LIN {X 0,Y 539.411,Z 297.162,A -85,B 0,C 180,E1 -4153.42,E2 -4153.42} C_VEL
LIN {X 0,Y 539.753,Z 202.979,A -85,B 0,C 180,E1 -4154.735,E2 -4154.735} C_VEL
LIN {X 0,Y 538.601,Z 196.337,A -85,B 0,C 180,E1 -4154.875,E2 -4154.875} C_VEL
LIN {X 0,Y 538.99,Z 174.234,A -85,B 0,C 180,E1 -4158.237,E2 -4158.237} C_VEL
LIN {X 0,Y 539.44,Z 154.956,A -85,B 0,C 180,E1 -4161.195,E2 -4161.195} C_VEL
LIN {X 0,Y 539.677,Z 143.31,A -85,B 0,C 180,E1 -4162.997,E2 -4162.997} C_VEL
LIN {X 0,Y 539.202,Z 140.592,A -85,B 0,C 180,E1 -4163.445,E2 -4163.445} C_VEL
LIN {X 0,Y 538.106,Z 138.749,A -85,B 0,C 180,E1 -4163.808,E2 -4163.808} C_VEL
LIN {X 0,Y 536.213,Z 137.465,A -85,B 0,C 180,E1 -4164.169,E2 -4164.169} C_VEL
LIN {X 0,Y 532.769,Z 136.298,A -85,B 0,C 180,E1 -4164.789,E2 -4164.789} C_VEL
LIN {X 0,Y 531.182,Z 135.998,A -85,B 0,C 180,E1 -4165.267,E2 -4165.267} C_VEL
LIN {X 0,Y 530.982,Z 135.97,A -85,B 0,C 180,E1 -4165.483,E2 -4165.483} C_VEL
LIN {X 0,Y 530.969,Z 135.967,A -85,B 0,C 180,E1 -4168.457,E2 -4168.457} C_VEL
LIN {X 0,Y 530.958,Z 135.972,A -85,B 0,C 180,E1 -4171.079,E2 -4171.079} C_VEL
LIN {X 0,Y 530.991,Z 135.967,A -85,B 0,C 180,E1 -4173.773,E2 -4173.773} C_VEL
LIN {X 0,Y 530.955,Z 135.968,A -85,B 0,C 180,E1 -4176.559,E2 -4176.559} C_VEL
LIN {X 0,Y 530.989,Z 135.966,A -85,B 0,C 180,E1 -4179.443,E2 -4179.443} C_VEL
LIN {X 0,Y 530.968,Z 135.967,A -85,B 0,C 180,E1 -4182.458,E2 -4182.458} C_VEL
LIN {X 0,Y 530.986,Z 135.965,A -85,B 0,C 180,E1 -4185.621,E2 -4185.621} C_VEL
LIN {X 0,Y 530.998,Z 135.966,A -85,B 0,C 180,E1 -4188.564,E2 -4188.564} C_VEL
LIN {X 0,Y 530.96,Z 135.97,A -85,B 0,C 180,E1 -4191.529,E2 -4191.529} C_VEL
LIN {X 0,Y 530.958,Z 135.972,A -85,B 0,C 180,E1 -4194.379,E2 -4194.379} C_VEL
LIN {X 0,Y 530.971,Z 135.971,A -85,B 0,C 180,E1 -4197.133,E2 -4197.133} C_VEL
LIN {X 0,Y 530.965,Z 135.968,A -85,B 0,C 180,E1 -4199.802,E2 -4199.802} C_VEL
LIN {X 0,Y 531.015,Z 135.969,A -85,B 0,C 180,E1 -4202.467,E2 -4202.467} C_VEL
LIN {X 0,Y 531.02,Z 136.091,A -85,B 0,C 180,E1 -4205.464,E2 -4205.464} C_VEL
LIN {X 0,Y 532.94,Z 145.226,A -85,B 0,C 180,E1 -4206.9,E2 -4206.9} C_VEL
LIN {X 0,Y 532.794,Z 159.001,A -85,B 0,C 180,E1 -4208.844,E2 -4208.844} C_VEL
LIN {X 0,Y 535.286,Z 169.811,A -85,B 0,C 180,E1 -4209.115,E2 -4209.115} C_VEL
LIN {X 0,Y 534.354,Z 324.425,A -85,B 0,C 180,E1 -4211.272,E2 -4211.272} C_VEL
LIN {X 0,Y 534.175,Z 339.836,A -85,B 0,C 180,E1 -4211.642,E2 -4211.642} C_VEL
LIN {X 0,Y 533.837,Z 353.957,A -85,B 0,C 180,E1 -4212.126,E2 -4212.126} C_VEL
LIN {X 0,Y 533.535,Z 367.904,A -85,B 0,C 180,E1 -4212.759,E2 -4212.759} C_VEL
LIN {X 0,Y 533.102,Z 381.485,A -85,B 0,C 180,E1 -4213.534,E2 -4213.534} C_VEL
LIN {X 0,Y 532.63,Z 394.075,A -85,B 0,C 180,E1 -4214.414,E2 -4214.414} C_VEL
LIN {X 0,Y 532.206,Z 406.499,A -85,B 0,C 180,E1 -4215.468,E2 -4215.468} C_VEL
LIN {X 0,Y 531.807,Z 417.877,A -85,B 0,C 180,E1 -4216.627,E2 -4216.627} C_VEL
LIN {X 0,Y 531.428,Z 427.452,A -85,B 0,C 180,E1 -4217.783,E2 -4217.783} C_VEL
LIN {X 0,Y 531.172,Z 436.798,A -85,B 0,C 180,E1 -4219.131,E2 -4219.131} C_VEL
LIN {X 0,Y 530.874,Z 444.587,A -85,B 0,C 180,E1 -4220.474,E2 -4220.474} C_VEL
LIN {X 0,Y 530.694,Z 451.826,A -85,B 0,C 180,E1 -4222.006,E2 -4222.006} C_VEL
LIN {X 0,Y 530.578,Z 457.254,A -85,B 0,C 180,E1 -4223.437,E2 -4223.437} C_VEL
LIN {X 0,Y 530.52,Z 460.953,A -85,B 0,C 180,E1 -4224.678,E2 -4224.678} C_VEL
LIN {X 0,Y 530.513,Z 464.408,A -85,B 0,C 180,E1 -4226.201,E2 -4226.201} C_VEL
LIN {X 0,Y 530.416,Z 466.698,A -85,B 0,C 180,E1 -4227.721,E2 -4227.721} C_VEL
LIN {X 0,Y 530.364,Z 467.866,A -85,B 0,C 180,E1 -4229.24,E2 -4229.24} C_VEL
LIN {X 0,Y 530.364,Z 467.884,A -85,B 0,C 180,E1 -4230.758,E2 -4230.758} C_VEL
LIN {X 0,Y 530.416,Z 466.787,A -85,B 0,C 180,E1 -4232.277,E2 -4232.277} C_VEL
LIN {X 0,Y 530.513,Z 464.572,A -85,B 0,C 180,E1 -4233.797,E2 -4233.797} C_VEL
LIN {X 0,Y 530.519,Z 461.201,A -85,B 0,C 180,E1 -4235.32,E2 -4235.32} C_VEL
LIN {X 0,Y 530.603,Z 456.572,A -85,B 0,C 180,E1 -4236.845,E2 -4236.845} C_VEL
LIN {X 0,Y 530.762,Z 450.558,A -85,B 0,C 180,E1 -4238.374,E2 -4238.374} C_VEL
LIN {X 0,Y 530.907,Z 442.996,A -85,B 0,C 180,E1 -4239.908,E2 -4239.908} C_VEL
LIN {X 0,Y 531.198,Z 434.918,A -85,B 0,C 180,E1 -4241.252,E2 -4241.252} C_VEL
LIN {X 0,Y 531.528,Z 425.173,A -85,B 0,C 180,E1 -4242.6,E2 -4242.6} C_VEL
LIN {X 0,Y 531.895,Z 415.216,A -85,B 0,C 180,E1 -4243.758,E2 -4243.758} C_VEL
LIN {X 0,Y 532.319,Z 403.281,A -85,B 0,C 180,E1 -4244.918,E2 -4244.918} C_VEL
LIN {X 0,Y 532.784,Z 391.316,A -85,B 0,C 180,E1 -4245.886,E2 -4245.886} C_VEL
LIN {X 0,Y 533.207,Z 378.321,A -85,B 0,C 180,E1 -4246.757,E2 -4246.757} C_VEL
LIN {X 0,Y 533.62,Z 363.9,A -85,B 0,C 180,E1 -4247.533,E2 -4247.533} C_VEL
LIN {X 0,Y 533.951,Z 350.087,A -85,B 0,C 180,E1 -4248.116,E2 -4248.116} C_VEL
LIN {X 0,Y 534.219,Z 334.867,A -85,B 0,C 180,E1 -4248.59,E2 -4248.59} C_VEL
LIN {X 0,Y 534.428,Z 319.25,A -85,B 0,C 180,E1 -4248.909,E2 -4248.909} C_VEL
LIN {X 0,Y 535.282,Z 170.427,A -85,B 0,C 180,E1 -4250.967,E2 -4250.967} C_VEL
LIN {X 0,Y 532.846,Z 159.131,A -85,B 0,C 180,E1 -4251.238,E2 -4251.238} C_VEL
LIN {X 0,Y 532.996,Z 145.964,A -85,B 0,C 180,E1 -4253.075,E2 -4253.075} C_VEL
LIN {X 0,Y 531.038,Z 135.963,A -85,B 0,C 180,E1 -4254.662,E2 -4254.662} C_VEL
LIN {X 0,Y 531.012,Z 135.968,A -85,B 0,C 180,E1 -4257.594,E2 -4257.594} C_VEL
LIN {X 0,Y 530.971,Z 135.968,A -85,B 0,C 180,E1 -4260.644,E2 -4260.644} C_VEL
LIN {X 0,Y 530.989,Z 135.969,A -85,B 0,C 180,E1 -4263.771,E2 -4263.771} C_VEL
LIN {X 0,Y 530.964,Z 135.967,A -85,B 0,C 180,E1 -4266.556,E2 -4266.556} C_VEL
LIN {X 0,Y 530.978,Z 135.96,A -85,B 0,C 180,E1 -4269.853,E2 -4269.853} C_VEL
LIN {X 0,Y 530.977,Z 135.965,A -85,B 0,C 180,E1 -4272.455,E2 -4272.455} C_VEL
LIN {X 0,Y 530.981,Z 135.969,A -85,B 0,C 180,E1 -4275.62,E2 -4275.62} C_VEL
LIN {X 0,Y 531,Z 135.962,A -85,B 0,C 180,E1 -4278.565,E2 -4278.565} C_VEL
LIN {X 0,Y 530.961,Z 135.972,A -85,B 0,C 180,E1 -4281.345,E2 -4281.345} C_VEL
LIN {X 0,Y 530.974,Z 135.965,A -85,B 0,C 180,E1 -4284.381,E2 -4284.381} C_VEL
LIN {X 0,Y 530.964,Z 135.974,A -85,B 0,C 180,E1 -4287.133,E2 -4287.133} C_VEL
LIN {X 0,Y 530.977,Z 135.96,A -85,B 0,C 180,E1 -4289.803,E2 -4289.803} C_VEL
LIN {X 0,Y 531.006,Z 135.962,A -85,B 0,C 180,E1 -4292.466,E2 -4292.466} C_VEL
LIN {X 0,Y 530.996,Z 135.966,A -85,B 0,C 180,E1 -4294.942,E2 -4294.942} C_VEL
LIN {X 0,Y 530.962,Z 135.967,A -85,B 0,C 180,E1 -4298.246,E2 -4298.246} C_VEL
LIN {X 0,Y 530.988,Z 135.965,A -85,B 0,C 180,E1 -4300.677,E2 -4300.677} C_VEL
LIN {X 0,Y 530.983,Z 135.971,A -85,B 0,C 180,E1 -4303.071,E2 -4303.071} C_VEL
LIN {X 0,Y 531.009,Z 135.96,A -85,B 0,C 180,E1 -4305.435,E2 -4305.435} C_VEL
LIN {X 0,Y 531.036,Z 135.958,A -85,B 0,C 180,E1 -4308.55,E2 -4308.55} C_VEL
LIN {X 0,Y 531.047,Z 135.954,A -85,B 0,C 180,E1 -4311.629,E2 -4311.629} C_VEL
LIN {X 0,Y 531.114,Z 135.949,A -85,B 0,C 180,E1 -4314.685,E2 -4314.685} C_VEL
LIN {X 0,Y 531.128,Z 135.945,A -85,B 0,C 180,E1 -4317.725,E2 -4317.725} C_VEL
LIN {X 0,Y 531.147,Z 135.946,A -85,B 0,C 180,E1 -4320.758,E2 -4320.758} C_VEL
LIN {X 0,Y 531.1,Z 135.952,A -85,B 0,C 180,E1 -4323.034,E2 -4323.034} C_VEL
LIN {X 0,Y 531.073,Z 135.951,A -85,B 0,C 180,E1 -4326.077,E2 -4326.077} C_VEL
LIN {X 0,Y 531.026,Z 135.959,A -85,B 0,C 180,E1 -4329.138,E2 -4329.138} C_VEL
LIN {X 0,Y 531.031,Z 135.96,A -85,B 0,C 180,E1 -4332.225,E2 -4332.225} C_VEL
LIN {X 0,Y 530.985,Z 135.962,A -85,B 0,C 180,E1 -4335.35,E2 -4335.35} C_VEL
LIN {X 0,Y 531.006,Z 135.959,A -85,B 0,C 180,E1 -4337.723,E2 -4337.723} C_VEL
LIN {X 0,Y 530.994,Z 135.964,A -85,B 0,C 180,E1 -4340.938,E2 -4340.938} C_VEL
LIN {X 0,Y 530.997,Z 135.964,A -85,B 0,C 180,E1 -4344.046,E2 -4344.046} C_VEL
LIN {X 0,Y 530.996,Z 135.965,A -85,B 0,C 180,E1 -4346.744,E2 -4346.744} C_VEL
LIN {X 0,Y 530.972,Z 135.961,A -85,B 0,C 180,E1 -4349.323,E2 -4349.323} C_VEL
LIN {X 0,Y 530.971,Z 135.972,A -85,B 0,C 180,E1 -4352.104,E2 -4352.104} C_VEL
LIN {X 0,Y 530.98,Z 135.964,A -85,B 0,C 180,E1 -4354.855,E2 -4354.855} C_VEL
LIN {X 0,Y 530.957,Z 135.968,A -85,B 0,C 180,E1 -4357.508,E2 -4357.508} C_VEL
LIN {X 0,Y 530.976,Z 135.959,A -85,B 0,C 180,E1 -4360.433,E2 -4360.433} C_VEL
LIN {X 0,Y 530.958,Z 135.967,A -85,B 0,C 180,E1 -4363.283,E2 -4363.283} C_VEL
LIN {X 0,Y 530.98,Z 135.968,A -85,B 0,C 180,E1 -4365.622,E2 -4365.622} C_VEL
LIN {X 0,Y 531,Z 135.964,A -85,B 0,C 180,E1 -4368.567,E2 -4368.567} C_VEL
LIN {X 0,Y 530.961,Z 135.967,A -85,B 0,C 180,E1 -4371.347,E2 -4371.347} C_VEL
LIN {X 0,Y 530.972,Z 135.966,A -85,B 0,C 180,E1 -4374.383,E2 -4374.383} C_VEL
LIN {X 0,Y 530.964,Z 135.967,A -85,B 0,C 180,E1 -4377.135,E2 -4377.135} C_VEL
LIN {X 0,Y 531.005,Z 136.164,A -85,B 0,C 180,E1 -4379.302,E2 -4379.302} C_VEL
LIN {X 0,Y 535.75,Z 152.052,A -85,B 0,C 180,E1 -4381.059,E2 -4381.059} C_VEL
LIN {X 0,Y 534.856,Z 180.096,A -85,B 0,C 180,E1 -4383.571,E2 -4383.571} C_VEL
LIN {X 0,Y 533.903,Z 213.965,A -85,B 0,C 180,E1 -4386.536,E2 -4386.536} C_VEL
LIN {X 0,Y 533.257,Z 242.128,A -85,B 0,C 180,E1 -4388.953,E2 -4388.953} C_VEL
LIN {X 0,Y 534.724,Z 254.825,A -85,B 0,C 180,E1 -4389.191,E2 -4389.191} C_VEL
LIN {X 0,Y 533.853,Z 410.343,A -85,B 0,C 180,E1 -4391.348,E2 -4391.348} C_VEL
LIN {X 0,Y 533.575,Z 426.116,A -85,B 0,C 180,E1 -4391.722,E2 -4391.722} C_VEL
LIN {X 0,Y 533.281,Z 441.621,A -85,B 0,C 180,E1 -4392.257,E2 -4392.257} C_VEL
LIN {X 0,Y 532.906,Z 454.584,A -85,B 0,C 180,E1 -4392.839,E2 -4392.839} C_VEL
LIN {X 0,Y 532.57,Z 468.468,A -85,B 0,C 180,E1 -4393.617,E2 -4393.617} C_VEL
LIN {X 0,Y 532.198,Z 481.236,A -85,B 0,C 180,E1 -4394.491,E2 -4394.491} C_VEL
LIN {X 0,Y 531.791,Z 494.19,A -85,B 0,C 180,E1 -4395.556,E2 -4395.556} C_VEL
LIN {X 0,Y 531.479,Z 505.043,A -85,B 0,C 180,E1 -4396.621,E2 -4396.621} C_VEL
LIN {X 0,Y 531.217,Z 515.097,A -85,B 0,C 180,E1 -4397.78,E2 -4397.78} C_VEL
LIN {X 0,Y 531.007,Z 524.955,A -85,B 0,C 180,E1 -4399.13,E2 -4399.13} C_VEL
LIN {X 0,Y 530.739,Z 533.148,A -85,B 0,C 180,E1 -4400.473,E2 -4400.473} C_VEL
LIN {X 0,Y 530.612,Z 540.805,A -85,B 0,C 180,E1 -4402.007,E2 -4402.007} C_VEL
LIN {X 0,Y 530.544,Z 546.617,A -85,B 0,C 180,E1 -4403.467,E2 -4403.467} C_VEL
LIN {X 0,Y 530.508,Z 550.371,A -85,B 0,C 180,E1 -4404.68,E2 -4404.68} C_VEL
LIN {X 0,Y 530.48,Z 553.888,A -85,B 0,C 180,E1 -4406.203,E2 -4406.203} C_VEL
LIN {X 0,Y 530.409,Z 556.19,A -85,B 0,C 180,E1 -4407.723,E2 -4407.723} C_VEL
LIN {X 0,Y 530.342,Z 557.348,A -85,B 0,C 180,E1 -4409.242,E2 -4409.242} C_VEL
LIN {X 0,Y 530.342,Z 557.346,A -85,B 0,C 180,E1 -4410.76,E2 -4410.76} C_VEL
LIN {X 0,Y 530.409,Z 556.183,A -85,B 0,C 180,E1 -4412.279,E2 -4412.279} C_VEL
LIN {X 0,Y 530.48,Z 553.879,A -85,B 0,C 180,E1 -4413.799,E2 -4413.799} C_VEL
LIN {X 0,Y 530.509,Z 550.368,A -85,B 0,C 180,E1 -4415.322,E2 -4415.322} C_VEL
LIN {X 0,Y 530.55,Z 545.488,A -85,B 0,C 180,E1 -4416.848,E2 -4416.848} C_VEL
LIN {X 0,Y 530.666,Z 539.044,A -85,B 0,C 180,E1 -4418.378,E2 -4418.378} C_VEL
LIN {X 0,Y 530.809,Z 530.894,A -85,B 0,C 180,E1 -4419.912,E2 -4419.912} C_VEL
LIN {X 0,Y 531.008,Z 522.208,A -85,B 0,C 180,E1 -4421.258,E2 -4421.258} C_VEL
LIN {X 0,Y 531.232,Z 513.345,A -85,B 0,C 180,E1 -4422.415,E2 -4422.415} C_VEL
LIN {X 0,Y 531.518,Z 502.89,A -85,B 0,C 180,E1 -4423.575,E2 -4423.575} C_VEL
LIN {X 0,Y 531.862,Z 490.44,A -85,B 0,C 180,E1 -4424.737,E2 -4424.737} C_VEL
LIN {X 0,Y 532.229,Z 477.975,A -85,B 0,C 180,E1 -4425.706,E2 -4425.706} C_VEL
LIN {X 0,Y 532.581,Z 464.402,A -85,B 0,C 180,E1 -4426.582,E2 -4426.582} C_VEL
LIN {X 0,Y 532.931,Z 450.475,A -85,B 0,C 180,E1 -4427.311,E2 -4427.311} C_VEL
LIN {X 0,Y 533.322,Z 436.416,A -85,B 0,C 180,E1 -4427.892,E2 -4427.892} C_VEL
LIN {X 0,Y 533.557,Z 421.573,A -85,B 0,C 180,E1 -4428.355,E2 -4428.355} C_VEL
LIN {X 0,Y 533.802,Z 405.468,A -85,B 0,C 180,E1 -4428.689,E2 -4428.689} C_VEL
LIN {X 0,Y 534.576,Z 252.777,A -85,B 0,C 180,E1 -4430.805,E2 -4430.805} C_VEL
LIN {X 0,Y 533.124,Z 241.458,A -85,B 0,C 180,E1 -4431.033,E2 -4431.033} C_VEL
LIN {X 0,Y 533.858,Z 208.007,A -85,B 0,C 180,E1 -4433.88,E2 -4433.88} C_VEL
LIN {X 0,Y 534.82,Z 174.765,A -85,B 0,C 180,E1 -4436.807,E2 -4436.807} C_VEL
LIN {X 0,Y 535.558,Z 151.471,A -85,B 0,C 180,E1 -4438.949,E2 -4438.949} C_VEL
LIN {X 0,Y 531.521,Z 137.946,A -85,B 0,C 180,E1 -4440.533,E2 -4440.533} C_VEL
LIN {X 0,Y 530.958,Z 135.974,A -85,B 0,C 180,E1 -4440.795,E2 -4440.795} C_VEL
LIN {X 0,Y 530.989,Z 135.973,A -85,B 0,C 180,E1 -4443.773,E2 -4443.773} C_VEL
LIN {X 0,Y 530.952,Z 135.971,A -85,B 0,C 180,E1 -4446.56,E2 -4446.56} C_VEL
LIN {X 0,Y 530.967,Z 135.974,A -85,B 0,C 180,E1 -4449.446,E2 -4449.446} C_VEL
LIN {X 0,Y 530.908,Z 135.976,A -85,B 0,C 180,E1 -4452.464,E2 -4452.464} C_VEL
LIN {X 0,Y 530.963,Z 135.974,A -85,B 0,C 180,E1 -4455.451,E2 -4455.451} C_VEL
LIN {X 0,Y 530.908,Z 135.976,A -85,B 0,C 180,E1 -4458.556,E2 -4458.556} C_VEL
LIN {X 0,Y 530.929,Z 135.977,A -85,B 0,C 180,E1 -4461.527,E2 -4461.527} C_VEL
LIN {X 0,Y 530.929,Z 135.975,A -85,B 0,C 180,E1 -4464.378,E2 -4464.378} C_VEL
LIN {X 0,Y 530.956,Z 135.975,A -85,B 0,C 180,E1 -4467.133,E2 -4467.133} C_VEL
LIN {X 0,Y 530.937,Z 135.973,A -85,B 0,C 180,E1 -4469.801,E2 -4469.801} C_VEL
LIN {X 0,Y 530.966,Z 135.974,A -85,B 0,C 180,E1 -4472.478,E2 -4472.478} C_VEL
LIN {X 0,Y 530.996,Z 136.108,A -85,B 0,C 180,E1 -4474.706,E2 -4474.706} C_VEL
LIN {X 0,Y 533.624,Z 147.119,A -85,B 0,C 180,E1 -4476.727,E2 -4476.727} C_VEL
LIN {X 0,Y 533.242,Z 162.09,A -85,B 0,C 180,E1 -4479.154,E2 -4479.154} C_VEL
LIN {X 0,Y 532.541,Z 182.09,A -85,B 0,C 180,E1 -4482.33,E2 -4482.33} C_VEL
LIN {X 0,Y 532.101,Z 198.36,A -85,B 0,C 180,E1 -4484.857,E2 -4484.857} C_VEL
LIN {X 0,Y 533.494,Z 205.069,A -85,B 0,C 180,E1 -4485.02,E2 -4485.02} C_VEL
LIN {X 0,Y 532.55,Z 309.27,A -85,B 0,C 180,E1 -4486.647,E2 -4486.647} C_VEL
LIN {X 0,Y 532.427,Z 323.125,A -85,B 0,C 180,E1 -4487.033,E2 -4487.033} C_VEL
LIN {X 0,Y 532.299,Z 335.189,A -85,B 0,C 180,E1 -4487.524,E2 -4487.524} C_VEL
LIN {X 0,Y 532.042,Z 347.599,A -85,B 0,C 180,E1 -4488.2,E2 -4488.2} C_VEL
LIN {X 0,Y 531.831,Z 358.421,A -85,B 0,C 180,E1 -4488.953,E2 -4488.953} C_VEL
LIN {X 0,Y 531.598,Z 367.373,A -85,B 0,C 180,E1 -4489.719,E2 -4489.719} C_VEL
LIN {X 0,Y 531.394,Z 376.557,A -85,B 0,C 180,E1 -4490.676,E2 -4490.676} C_VEL
LIN {X 0,Y 531.17,Z 385.415,A -85,B 0,C 180,E1 -4491.823,E2 -4491.823} C_VEL
LIN {X 0,Y 530.97,Z 393.171,A -85,B 0,C 180,E1 -4493.081,E2 -4493.081} C_VEL
LIN {X 0,Y 530.872,Z 399.015,A -85,B 0,C 180,E1 -4494.302,E2 -4494.302} C_VEL
LIN {X 0,Y 530.776,Z 403.281,A -85,B 0,C 180,E1 -4495.443,E2 -4495.443} C_VEL
LIN {X 0,Y 530.715,Z 405.526,A -85,B 0,C 180,E1 -4496.204,E2 -4496.204} C_VEL
LIN {X 0,Y 530.672,Z 407.347,A -85,B 0,C 180,E1 -4496.963,E2 -4496.963} C_VEL
LIN {X 0,Y 530.635,Z 408.728,A -85,B 0,C 180,E1 -4497.723,E2 -4497.723} C_VEL
LIN {X 0,Y 530.614,Z 410.27,A -85,B 0,C 180,E1 -4499.241,E2 -4499.241} C_VEL
LIN {X 0,Y 530.604,Z 410.472,A -85,B 0,C 180,E1 -4500,E2 -4500} C_VEL
LIN {X 0,Y 530.612,Z 410.264,A -85,B 0,C 180,E1 -4500.759,E2 -4500.759} C_VEL
LIN {X 0,Y 530.577,Z 409.667,A -85,B 0,C 180,E1 -4501.518,E2 -4501.518} C_VEL
LIN {X 0,Y 530.634,Z 408.666,A -85,B 0,C 180,E1 -4502.277,E2 -4502.277} C_VEL
LIN {X 0,Y 530.639,Z 407.284,A -85,B 0,C 180,E1 -4503.037,E2 -4503.037} C_VEL
LIN {X 0,Y 530.743,Z 404.377,A -85,B 0,C 180,E1 -4504.177,E2 -4504.177} C_VEL
LIN {X 0,Y 530.686,Z 400.478,A -85,B 0,C 180,E1 -4505.319,E2 -4505.319} C_VEL
LIN {X 0,Y 530.873,Z 394.539,A -85,B 0,C 180,E1 -4506.635,E2 -4506.635} C_VEL
LIN {X 0,Y 530.997,Z 387.854,A -85,B 0,C 180,E1 -4507.797,E2 -4507.797} C_VEL
LIN {X 0,Y 531.183,Z 379.638,A -85,B 0,C 180,E1 -4508.944,E2 -4508.944} C_VEL
LIN {X 0,Y 531.398,Z 371.215,A -85,B 0,C 180,E1 -4509.9,E2 -4509.9} C_VEL
LIN {X 0,Y 531.669,Z 360.803,A -85,B 0,C 180,E1 -4510.858,E2 -4510.858} C_VEL
LIN {X 0,Y 531.879,Z 349.43,A -85,B 0,C 180,E1 -4511.697,E2 -4511.697} C_VEL
LIN {X 0,Y 532.117,Z 337.327,A -85,B 0,C 180,E1 -4512.394,E2 -4512.394} C_VEL
LIN {X 0,Y 532.185,Z 325.161,A -85,B 0,C 180,E1 -4512.925,E2 -4512.925} C_VEL
LIN {X 0,Y 532.43,Z 311.946,A -85,B 0,C 180,E1 -4513.332,E2 -4513.332} C_VEL
LIN {X 0,Y 532.537,Z 297.536,A -85,B 0,C 180,E1 -4513.596,E2 -4513.596} C_VEL
LIN {X 0,Y 532.952,Z 203.638,A -85,B 0,C 180,E1 -4514.942,E2 -4514.942} C_VEL
LIN {X 0,Y 531.632,Z 196.503,A -85,B 0,C 180,E1 -4515.111,E2 -4515.111} C_VEL
LIN {X 0,Y 532.104,Z 174.496,A -85,B 0,C 180,E1 -4518.481,E2 -4518.481} C_VEL
LIN {X 0,Y 532.553,Z 156.431,A -85,B 0,C 180,E1 -4521.279,E2 -4521.279} C_VEL
LIN {X 0,Y 532.784,Z 144.765,A -85,B 0,C 180,E1 -4523.106,E2 -4523.106} C_VEL
LIN {X 0,Y 531.007,Z 135.967,A -85,B 0,C 180,E1 -4524.614,E2 -4524.614} C_VEL
LIN {X 0,Y 530.982,Z 135.97,A -85,B 0,C 180,E1 -4525.483,E2 -4525.483} C_VEL
LIN {X 0,Y 530.302,Z 136.056,A -85,B 0,C 180,E1 -4526.117,E2 -4526.117} C_VEL
LIN {X 0,Y 527.417,Z 136.415,A -85,B 0,C 180,E1 -4527.145,E2 -4527.145} C_VEL
LIN {X 0,Y 525.003,Z 136.714,A -85,B 0,C 180,E1 -4527.973,E2 -4527.973} C_VEL
LIN {X 0,Y 523.994,Z 136.837,A -85,B 0,C 180,E1 -4528.612,E2 -4528.612} C_VEL
LIN {X 0,Y 523.927,Z 136.846,A -85,B 0,C 180,E1 -4528.829,E2 -4528.829} C_VEL
LIN {X 0,Y 523.924,Z 136.851,A -85,B 0,C 180,E1 -4531.544,E2 -4531.544} C_VEL
LIN {X 0,Y 523.936,Z 136.842,A -85,B 0,C 180,E1 -4534.29,E2 -4534.29} C_VEL
LIN {X 0,Y 523.909,Z 136.853,A -85,B 0,C 180,E1 -4537.132,E2 -4537.132} C_VEL
LIN {X 0,Y 523.943,Z 136.838,A -85,B 0,C 180,E1 -4540.13,E2 -4540.13} C_VEL
LIN {X 0,Y 523.906,Z 136.85,A -85,B 0,C 180,E1 -4543.169,E2 -4543.169} C_VEL
LIN {X 0,Y 523.94,Z 136.842,A -85,B 0,C 180,E1 -4545.771,E2 -4545.771} C_VEL
LIN {X 0,Y 523.944,Z 136.85,A -85,B 0,C 180,E1 -4548.907,E2 -4548.907} C_VEL
LIN {X 0,Y 523.919,Z 136.846,A -85,B 0,C 180,E1 -4551.898,E2 -4551.898} C_VEL
LIN {X 0,Y 523.928,Z 136.85,A -85,B 0,C 180,E1 -4554.911,E2 -4554.911} C_VEL
LIN {X 0,Y 523.939,Z 136.843,A -85,B 0,C 180,E1 -4557.679,E2 -4557.679} C_VEL
LIN {X 0,Y 523.957,Z 136.847,A -85,B 0,C 180,E1 -4560.676,E2 -4560.676} C_VEL
LIN {X 0,Y 523.978,Z 136.84,A -85,B 0,C 180,E1 -4563.728,E2 -4563.728} C_VEL
LIN {X 0,Y 524.002,Z 136.936,A -85,B 0,C 180,E1 -4565.22,E2 -4565.22} C_VEL
LIN {X 0,Y 526.076,Z 146.848,A -85,B 0,C 180,E1 -4566.79,E2 -4566.79} C_VEL
LIN {X 0,Y 525.983,Z 159.147,A -85,B 0,C 180,E1 -4568.53,E2 -4568.53} C_VEL
LIN {X 0,Y 526.485,Z 161.494,A -85,B 0,C 180,E1 -4568.619,E2 -4568.619} C_VEL
LIN {X 0,Y 528.662,Z 170.75,A -85,B 0,C 180,E1 -4568.847,E2 -4568.847} C_VEL
LIN {X 0,Y 527.68,Z 324.547,A -85,B 0,C 180,E1 -4571.019,E2 -4571.019} C_VEL
LIN {X 0,Y 527.466,Z 339.514,A -85,B 0,C 180,E1 -4571.375,E2 -4571.375} C_VEL
LIN {X 0,Y 527.152,Z 353.273,A -85,B 0,C 180,E1 -4571.841,E2 -4571.841} C_VEL
LIN {X 0,Y 526.837,Z 366.567,A -85,B 0,C 180,E1 -4572.432,E2 -4572.432} C_VEL
LIN {X 0,Y 526.42,Z 379.002,A -85,B 0,C 180,E1 -4573.119,E2 -4573.119} C_VEL
LIN {X 0,Y 525.99,Z 392.139,A -85,B 0,C 180,E1 -4574.014,E2 -4574.014} C_VEL
LIN {X 0,Y 525.484,Z 403.914,A -85,B 0,C 180,E1 -4574.981,E2 -4574.981} C_VEL
LIN {X 0,Y 525.043,Z 414.905,A -85,B 0,C 180,E1 -4576.057,E2 -4576.057} C_VEL
LIN {X 0,Y 524.631,Z 425.012,A -85,B 0,C 180,E1 -4577.229,E2 -4577.229} C_VEL
LIN {X 0,Y 524.246,Z 434.882,A -85,B 0,C 180,E1 -4578.594,E2 -4578.594} C_VEL
LIN {X 0,Y 523.933,Z 443.072,A -85,B 0,C 180,E1 -4579.956,E2 -4579.956} C_VEL
LIN {X 0,Y 523.741,Z 450.731,A -85,B 0,C 180,E1 -4581.511,E2 -4581.511} C_VEL
LIN {X 0,Y 523.563,Z 456.826,A -85,B 0,C 180,E1 -4583.06,E2 -4583.06} C_VEL
LIN {X 0,Y 523.468,Z 461.539,A -85,B 0,C 180,E1 -4584.606,E2 -4584.606} C_VEL
LIN {X 0,Y 523.466,Z 464.992,A -85,B 0,C 180,E1 -4586.15,E2 -4586.15} C_VEL
LIN {X 0,Y 523.344,Z 467.283,A -85,B 0,C 180,E1 -4587.69,E2 -4587.69} C_VEL
LIN {X 0,Y 523.289,Z 468.451,A -85,B 0,C 180,E1 -4589.229,E2 -4589.229} C_VEL
LIN {X 0,Y 523.289,Z 468.469,A -85,B 0,C 180,E1 -4590.769,E2 -4590.769} C_VEL
LIN {X 0,Y 523.344,Z 467.371,A -85,B 0,C 180,E1 -4592.308,E2 -4592.308} C_VEL
LIN {X 0,Y 523.466,Z 465.154,A -85,B 0,C 180,E1 -4593.848,E2 -4593.848} C_VEL
LIN {X 0,Y 523.466,Z 461.784,A -85,B 0,C 180,E1 -4595.392,E2 -4595.392} C_VEL
LIN {X 0,Y 523.561,Z 457.155,A -85,B 0,C 180,E1 -4596.938,E2 -4596.938} C_VEL
LIN {X 0,Y 523.736,Z 451.14,A -85,B 0,C 180,E1 -4598.487,E2 -4598.487} C_VEL
LIN {X 0,Y 523.922,Z 443.574,A -85,B 0,C 180,E1 -4600.042,E2 -4600.042} C_VEL
LIN {X 0,Y 524.237,Z 435.494,A -85,B 0,C 180,E1 -4601.404,E2 -4601.404} C_VEL
LIN {X 0,Y 524.604,Z 425.746,A -85,B 0,C 180,E1 -4602.769,E2 -4602.769} C_VEL
LIN {X 0,Y 525.007,Z 415.784,A -85,B 0,C 180,E1 -4603.942,E2 -4603.942} C_VEL
LIN {X 0,Y 525.477,Z 403.843,A -85,B 0,C 180,E1 -4605.117,E2 -4605.117} C_VEL
LIN {X 0,Y 525.982,Z 391.733,A -85,B 0,C 180,E1 -4606.107,E2 -4606.107} C_VEL
LIN {X 0,Y 526.453,Z 378.863,A -85,B 0,C 180,E1 -4606.978,E2 -4606.978} C_VEL
LIN {X 0,Y 526.895,Z 364.425,A -85,B 0,C 180,E1 -4607.764,E2 -4607.764} C_VEL
LIN {X 0,Y 527.242,Z 350.592,A -85,B 0,C 180,E1 -4608.354,E2 -4608.354} C_VEL
LIN {X 0,Y 527.529,Z 334.985,A -85,B 0,C 180,E1 -4608.843,E2 -4608.843} C_VEL
LIN {X 0,Y 527.742,Z 320.503,A -85,B 0,C 180,E1 -4609.144,E2 -4609.144} C_VEL
LIN {X 0,Y 528.667,Z 170.847,A -85,B 0,C 180,E1 -4611.242,E2 -4611.242} C_VEL
LIN {X 0,Y 526.036,Z 159.447,A -85,B 0,C 180,E1 -4611.525,E2 -4611.525} C_VEL
LIN {X 0,Y 526.137,Z 147.411,A -85,B 0,C 180,E1 -4613.205,E2 -4613.205} C_VEL
LIN {X 0,Y 523.982,Z 136.843,A -85,B 0,C 180,E1 -4614.912,E2 -4614.912} C_VEL
LIN {X 0,Y 523.966,Z 136.843,A -85,B 0,C 180,E1 -4617.998,E2 -4617.998} C_VEL
LIN {X 0,Y 523.944,Z 136.845,A -85,B 0,C 180,E1 -4620.854,E2 -4620.854} C_VEL
LIN {X 0,Y 523.959,Z 136.845,A -85,B 0,C 180,E1 -4623.734,E2 -4623.734} C_VEL
LIN {X 0,Y 523.918,Z 136.844,A -85,B 0,C 180,E1 -4626.403,E2 -4626.403} C_VEL
LIN {X 0,Y 523.918,Z 136.849,A -85,B 0,C 180,E1 -4629.083,E2 -4629.083} C_VEL
LIN {X 0,Y 523.951,Z 136.841,A -85,B 0,C 180,E1 -4632.117,E2 -4632.117} C_VEL
LIN {X 0,Y 523.949,Z 136.847,A -85,B 0,C 180,E1 -4635.308,E2 -4635.308} C_VEL
LIN {X 0,Y 523.965,Z 136.839,A -85,B 0,C 180,E1 -4638.687,E2 -4638.687} C_VEL
LIN {X 0,Y 523.946,Z 136.846,A -85,B 0,C 180,E1 -4641.075,E2 -4641.075} C_VEL
LIN {X 0,Y 523.92,Z 136.844,A -85,B 0,C 180,E1 -4643.827,E2 -4643.827} C_VEL
LIN {X 0,Y 523.934,Z 136.842,A -85,B 0,C 180,E1 -4646.635,E2 -4646.635} C_VEL
LIN {X 0,Y 523.955,Z 136.839,A -85,B 0,C 180,E1 -4649.356,E2 -4649.356} C_VEL
LIN {X 0,Y 523.97,Z 136.838,A -85,B 0,C 180,E1 -4652.28,E2 -4652.28} C_VEL
LIN {X 0,Y 523.943,Z 136.842,A -85,B 0,C 180,E1 -4654.581,E2 -4654.581} C_VEL
LIN {X 0,Y 523.907,Z 136.853,A -85,B 0,C 180,E1 -4657.106,E2 -4657.106} C_VEL
LIN {X 0,Y 523.969,Z 136.835,A -85,B 0,C 180,E1 -4659.865,E2 -4659.865} C_VEL
LIN {X 0,Y 523.961,Z 136.843,A -85,B 0,C 180,E1 -4662.837,E2 -4662.837} C_VEL
LIN {X 0,Y 523.966,Z 136.839,A -85,B 0,C 180,E1 -4665.235,E2 -4665.235} C_VEL
LIN {X 0,Y 524.001,Z 136.832,A -85,B 0,C 180,E1 -4668.394,E2 -4668.394} C_VEL
LIN {X 0,Y 523.995,Z 136.833,A -85,B 0,C 180,E1 -4671.516,E2 -4671.516} C_VEL
LIN {X 0,Y 524.075,Z 136.824,A -85,B 0,C 180,E1 -4674.614,E2 -4674.614} C_VEL
LIN {X 0,Y 524.101,Z 136.821,A -85,B 0,C 180,E1 -4677.694,E2 -4677.694} C_VEL
LIN {X 0,Y 524.116,Z 136.821,A -85,B 0,C 180,E1 -4680.768,E2 -4680.768} C_VEL
LIN {X 0,Y 524.066,Z 136.828,A -85,B 0,C 180,E1 -4683.075,E2 -4683.075} C_VEL
LIN {X 0,Y 524.035,Z 136.828,A -85,B 0,C 180,E1 -4686.159,E2 -4686.159} C_VEL
LIN {X 0,Y 523.994,Z 136.834,A -85,B 0,C 180,E1 -4689.262,E2 -4689.262} C_VEL
LIN {X 0,Y 523.997,Z 136.831,A -85,B 0,C 180,E1 -4691.743,E2 -4691.743} C_VEL
LIN {X 0,Y 523.982,Z 136.836,A -85,B 0,C 180,E1 -4695.053,E2 -4695.053} C_VEL
LIN {X 0,Y 523.954,Z 136.839,A -85,B 0,C 180,E1 -4697.969,E2 -4697.969} C_VEL
LIN {X 0,Y 523.963,Z 136.842,A -85,B 0,C 180,E1 -4700.41,E2 -4700.41} C_VEL
LIN {X 0,Y 523.934,Z 136.842,A -85,B 0,C 180,E1 -4702.892,E2 -4702.892} C_VEL
LIN {X 0,Y 523.974,Z 136.838,A -85,B 0,C 180,E1 -4706.02,E2 -4706.02} C_VEL
LIN {X 0,Y 523.93,Z 136.84,A -85,B 0,C 180,E1 -4708.875,E2 -4708.875} C_VEL
LIN {X 0,Y 523.921,Z 136.844,A -85,B 0,C 180,E1 -4711.544,E2 -4711.544} C_VEL
LIN {X 0,Y 523.935,Z 136.846,A -85,B 0,C 180,E1 -4714.29,E2 -4714.29} C_VEL
LIN {X 0,Y 523.902,Z 136.845,A -85,B 0,C 180,E1 -4717.133,E2 -4717.133} C_VEL
LIN {X 0,Y 523.928,Z 136.836,A -85,B 0,C 180,E1 -4720.131,E2 -4720.131} C_VEL
LIN {X 0,Y 523.929,Z 136.846,A -85,B 0,C 180,E1 -4722.46,E2 -4722.46} C_VEL
LIN {X 0,Y 523.948,Z 136.841,A -85,B 0,C 180,E1 -4725.31,E2 -4725.31} C_VEL
LIN {X 0,Y 523.965,Z 136.84,A -85,B 0,C 180,E1 -4728.689,E2 -4728.689} C_VEL
LIN {X 0,Y 523.918,Z 136.843,A -85,B 0,C 180,E1 -4731.08,E2 -4731.08} C_VEL
LIN {X 0,Y 523.92,Z 136.849,A -85,B 0,C 180,E1 -4733.828,E2 -4733.828} C_VEL
LIN {X 0,Y 523.936,Z 136.842,A -85,B 0,C 180,E1 -4736.637,E2 -4736.637} C_VEL
LIN {X 0,Y 523.923,Z 136.906,A -85,B 0,C 180,E1 -4738.959,E2 -4738.959} C_VEL
LIN {X 0,Y 529.084,Z 154.102,A -85,B 0,C 180,E1 -4740.891,E2 -4740.891} C_VEL
LIN {X 0,Y 528.2,Z 179.45,A -85,B 0,C 180,E1 -4743.198,E2 -4743.198} C_VEL
LIN {X 0,Y 527.137,Z 213.347,A -85,B 0,C 180,E1 -4746.216,E2 -4746.216} C_VEL
LIN {X 0,Y 526.366,Z 241.865,A -85,B 0,C 180,E1 -4748.704,E2 -4748.704} C_VEL
LIN {X 0,Y 527.974,Z 255.236,A -85,B 0,C 180,E1 -4748.96,E2 -4748.96} C_VEL
LIN {X 0,Y 527,Z 409.198,A -85,B 0,C 180,E1 -4751.133,E2 -4751.133} C_VEL
LIN {X 0,Y 526.718,Z 424.798,A -85,B 0,C 180,E1 -4751.502,E2 -4751.502} C_VEL
LIN {X 0,Y 526.377,Z 439.927,A -85,B 0,C 180,E1 -4752.02,E2 -4752.02} C_VEL
LIN {X 0,Y 525.947,Z 454.96,A -85,B 0,C 180,E1 -4752.705,E2 -4752.705} C_VEL
LIN {X 0,Y 525.581,Z 468.637,A -85,B 0,C 180,E1 -4753.493,E2 -4753.493} C_VEL
LIN {X 0,Y 525.131,Z 482.52,A -85,B 0,C 180,E1 -4754.476,E2 -4754.476} C_VEL
LIN {X 0,Y 524.701,Z 495.119,A -85,B 0,C 180,E1 -4755.555,E2 -4755.555} C_VEL
LIN {X 0,Y 524.36,Z 507.463,A -85,B 0,C 180,E1 -4756.831,E2 -4756.831} C_VEL
LIN {X 0,Y 524.031,Z 518.075,A -85,B 0,C 180,E1 -4758.146,E2 -4758.146} C_VEL
LIN {X 0,Y 523.853,Z 527.621,A -85,B 0,C 180,E1 -4759.566,E2 -4759.566} C_VEL
LIN {X 0,Y 523.643,Z 534.212,A -85,B 0,C 180,E1 -4760.733,E2 -4760.733} C_VEL
LIN {X 0,Y 523.514,Z 541.479,A -85,B 0,C 180,E1 -4762.286,E2 -4762.286} C_VEL
LIN {X 0,Y 523.483,Z 547.198,A -85,B 0,C 180,E1 -4763.835,E2 -4763.835} C_VEL
LIN {X 0,Y 523.354,Z 551.504,A -85,B 0,C 180,E1 -4765.38,E2 -4765.38} C_VEL
LIN {X 0,Y 523.388,Z 554.536,A -85,B 0,C 180,E1 -4766.922,E2 -4766.922} C_VEL
LIN {X 0,Y 523.282,Z 556.325,A -85,B 0,C 180,E1 -4768.462,E2 -4768.462} C_VEL
LIN {X 0,Y 523.263,Z 556.936,A -85,B 0,C 180,E1 -4770.001,E2 -4770.001} C_VEL
LIN {X 0,Y 523.283,Z 556.314,A -85,B 0,C 180,E1 -4771.54,E2 -4771.54} C_VEL
LIN {X 0,Y 523.388,Z 554.51,A -85,B 0,C 180,E1 -4773.08,E2 -4773.08} C_VEL
LIN {X 0,Y 523.374,Z 551.464,A -85,B 0,C 180,E1 -4774.622,E2 -4774.622} C_VEL
LIN {X 0,Y 523.471,Z 547.132,A -85,B 0,C 180,E1 -4776.167,E2 -4776.167} C_VEL
LIN {X 0,Y 523.54,Z 541.371,A -85,B 0,C 180,E1 -4777.716,E2 -4777.716} C_VEL
LIN {X 0,Y 523.668,Z 534.032,A -85,B 0,C 180,E1 -4779.269,E2 -4779.269} C_VEL
LIN {X 0,Y 523.885,Z 526.18,A -85,B 0,C 180,E1 -4780.63,E2 -4780.63} C_VEL
LIN {X 0,Y 524.058,Z 516.982,A -85,B 0,C 180,E1 -4781.959,E2 -4781.959} C_VEL
LIN {X 0,Y 524.347,Z 506.985,A -85,B 0,C 180,E1 -4783.172,E2 -4783.172} C_VEL
LIN {X 0,Y 524.723,Z 494.488,A -85,B 0,C 180,E1 -4784.446,E2 -4784.446} C_VEL
LIN {X 0,Y 525.097,Z 481.694,A -85,B 0,C 180,E1 -4785.527,E2 -4785.527} C_VEL
LIN {X 0,Y 525.458,Z 469.068,A -85,B 0,C 180,E1 -4786.413,E2 -4786.413} C_VEL
LIN {X 0,Y 525.85,Z 455.458,A -85,B 0,C 180,E1 -4787.2,E2 -4787.2} C_VEL
LIN {X 0,Y 526.238,Z 441.702,A -85,B 0,C 180,E1 -4787.839,E2 -4787.839} C_VEL
LIN {X 0,Y 526.567,Z 426.821,A -85,B 0,C 180,E1 -4788.372,E2 -4788.372} C_VEL
LIN {X 0,Y 526.82,Z 412.043,A -85,B 0,C 180,E1 -4788.75,E2 -4788.75} C_VEL
LIN {X 0,Y 526.924,Z 391.379,A -85,B 0,C 180,E1 -4789.074,E2 -4789.074} C_VEL
LIN {X 0,Y 527.778,Z 263.989,A -85,B 0,C 180,E1 -4790.869,E2 -4790.869} C_VEL
LIN {X 0,Y 527.686,Z 252.778,A -85,B 0,C 180,E1 -4791.036,E2 -4791.036} C_VEL
LIN {X 0,Y 526.21,Z 241.048,A -85,B 0,C 180,E1 -4791.276,E2 -4791.276} C_VEL
LIN {X 0,Y 527.043,Z 208.414,A -85,B 0,C 180,E1 -4794.104,E2 -4794.104} C_VEL
LIN {X 0,Y 528.161,Z 175.205,A -85,B 0,C 180,E1 -4797.092,E2 -4797.092} C_VEL
LIN {X 0,Y 528.971,Z 153.674,A -85,B 0,C 180,E1 -4799.118,E2 -4799.118} C_VEL
LIN {X 0,Y 524.714,Z 139.415,A -85,B 0,C 180,E1 -4800.847,E2 -4800.847} C_VEL
LIN {X 0,Y 523.925,Z 136.849,A -85,B 0,C 180,E1 -4801.208,E2 -4801.208} C_VEL
LIN {X 0,Y 523.933,Z 136.85,A -85,B 0,C 180,E1 -4804.291,E2 -4804.291} C_VEL
LIN {X 0,Y 523.906,Z 136.85,A -85,B 0,C 180,E1 -4807.133,E2 -4807.133} C_VEL
LIN {X 0,Y 523.916,Z 136.849,A -85,B 0,C 180,E1 -4810.127,E2 -4810.127} C_VEL
LIN {X 0,Y 523.874,Z 136.856,A -85,B 0,C 180,E1 -4813.173,E2 -4813.173} C_VEL
LIN {X 0,Y 523.919,Z 136.85,A -85,B 0,C 180,E1 -4815.77,E2 -4815.77} C_VEL
LIN {X 0,Y 523.854,Z 136.858,A -85,B 0,C 180,E1 -4818.9,E2 -4818.9} C_VEL
LIN {X 0,Y 523.889,Z 136.851,A -85,B 0,C 180,E1 -4821.896,E2 -4821.896} C_VEL
LIN {X 0,Y 523.916,Z 136.853,A -85,B 0,C 180,E1 -4824.914,E2 -4824.914} C_VEL
LIN {X 0,Y 523.904,Z 136.85,A -85,B 0,C 180,E1 -4827.686,E2 -4827.686} C_VEL
LIN {X 0,Y 523.934,Z 136.85,A -85,B 0,C 180,E1 -4830.682,E2 -4830.682} C_VEL
LIN {X 0,Y 523.906,Z 136.855,A -85,B 0,C 180,E1 -4833.725,E2 -4833.725} C_VEL
LIN {X 0,Y 523.95,Z 137.025,A -85,B 0,C 180,E1 -4834.318,E2 -4834.318} C_VEL
LIN {X 0,Y 526.651,Z 148.064,A -85,B 0,C 180,E1 -4836.401,E2 -4836.401} C_VEL
LIN {X 0,Y 526.977,Z 151.255,A -85,B 0,C 180,E1 -4836.959,E2 -4836.959} C_VEL
LIN {X 0,Y 526.244,Z 169.224,A -85,B 0,C 180,E1 -4839.886,E2 -4839.886} C_VEL
LIN {X 0,Y 525.569,Z 189.212,A -85,B 0,C 180,E1 -4843.092,E2 -4843.092} C_VEL
LIN {X 0,Y 525.234,Z 198.691,A -85,B 0,C 180,E1 -4844.588,E2 -4844.588} C_VEL
LIN {X 0,Y 526.725,Z 205.202,A -85,B 0,C 180,E1 -4844.765,E2 -4844.765} C_VEL
LIN {X 0,Y 525.694,Z 310.241,A -85,B 0,C 180,E1 -4846.47,E2 -4846.47} C_VEL
LIN {X 0,Y 525.567,Z 324.007,A -85,B 0,C 180,E1 -4846.86,E2 -4846.86} C_VEL
LIN {X 0,Y 525.435,Z 336.069,A -85,B 0,C 180,E1 -4847.358,E2 -4847.358} C_VEL
LIN {X 0,Y 525.163,Z 348.53,A -85,B 0,C 180,E1 -4848.046,E2 -4848.046} C_VEL
LIN {X 0,Y 524.929,Z 359.323,A -85,B 0,C 180,E1 -4848.806,E2 -4848.806} C_VEL
LIN {X 0,Y 524.688,Z 368.296,A -85,B 0,C 180,E1 -4849.582,E2 -4849.582} C_VEL
LIN {X 0,Y 524.464,Z 377.511,A -85,B 0,C 180,E1 -4850.552,E2 -4850.552} C_VEL
LIN {X 0,Y 524.218,Z 386.391,A -85,B 0,C 180,E1 -4851.714,E2 -4851.714} C_VEL
LIN {X 0,Y 523.994,Z 394.168,A -85,B 0,C 180,E1 -4852.989,E2 -4852.989} C_VEL
LIN {X 0,Y 523.891,Z 400.024,A -85,B 0,C 180,E1 -4854.226,E2 -4854.226} C_VEL
LIN {X 0,Y 523.772,Z 404.298,A -85,B 0,C 180,E1 -4855.382,E2 -4855.382} C_VEL
LIN {X 0,Y 523.704,Z 406.544,A -85,B 0,C 180,E1 -4856.153,E2 -4856.153} C_VEL
LIN {X 0,Y 523.656,Z 408.365,A -85,B 0,C 180,E1 -4856.923,E2 -4856.923} C_VEL
LIN {X 0,Y 523.625,Z 409.744,A -85,B 0,C 180,E1 -4857.692,E2 -4857.692} C_VEL
LIN {X 0,Y 523.602,Z 411.271,A -85,B 0,C 180,E1 -4859.231,E2 -4859.231} C_VEL
LIN {X 0,Y 523.589,Z 411.466,A -85,B 0,C 180,E1 -4860,E2 -4860} C_VEL
LIN {X 0,Y 523.599,Z 411.248,A -85,B 0,C 180,E1 -4860.769,E2 -4860.769} C_VEL
LIN {X 0,Y 523.622,Z 409.616,A -85,B 0,C 180,E1 -4862.308,E2 -4862.308} C_VEL
LIN {X 0,Y 523.611,Z 408.224,A -85,B 0,C 180,E1 -4863.078,E2 -4863.078} C_VEL
LIN {X 0,Y 523.73,Z 405.286,A -85,B 0,C 180,E1 -4864.233,E2 -4864.233} C_VEL
LIN {X 0,Y 523.679,Z 401.355,A -85,B 0,C 180,E1 -4865.391,E2 -4865.391} C_VEL
LIN {X 0,Y 523.883,Z 395.874,A -85,B 0,C 180,E1 -4866.627,E2 -4866.627} C_VEL
LIN {X 0,Y 524.026,Z 388.64,A -85,B 0,C 180,E1 -4867.901,E2 -4867.901} C_VEL
LIN {X 0,Y 524.204,Z 380.388,A -85,B 0,C 180,E1 -4869.064,E2 -4869.064} C_VEL
LIN {X 0,Y 524.453,Z 371.921,A -85,B 0,C 180,E1 -4870.033,E2 -4870.033} C_VEL
LIN {X 0,Y 524.729,Z 362.627,A -85,B 0,C 180,E1 -4870.905,E2 -4870.905} C_VEL
LIN {X 0,Y 524.953,Z 352.038,A -85,B 0,C 180,E1 -4871.716,E2 -4871.716} C_VEL
LIN {X 0,Y 525.167,Z 339.771,A -85,B 0,C 180,E1 -4872.462,E2 -4872.462} C_VEL
LIN {X 0,Y 525.339,Z 328.238,A -85,B 0,C 180,E1 -4872.998,E2 -4872.998} C_VEL
LIN {X 0,Y 525.505,Z 315.104,A -85,B 0,C 180,E1 -4873.437,E2 -4873.437} C_VEL
LIN {X 0,Y 525.625,Z 302.706,A -85,B 0,C 180,E1 -4873.705,E2 -4873.705} C_VEL
LIN {X 0,Y 526.174,Z 204.694,A -85,B 0,C 180,E1 -4875.149,E2 -4875.149} C_VEL
LIN {X 0,Y 524.703,Z 196.769,A -85,B 0,C 180,E1 -4875.336,E2 -4875.336} C_VEL
LIN {X 0,Y 525.178,Z 175.986,A -85,B 0,C 180,E1 -4878.545,E2 -4878.545} C_VEL
LIN {X 0,Y 525.656,Z 157.943,A -85,B 0,C 180,E1 -4881.367,E2 -4881.367} C_VEL
LIN {X 0,Y 525.895,Z 146.217,A -85,B 0,C 180,E1 -4883.218,E2 -4883.218} C_VEL
LIN {X 0,Y 523.991,Z 136.842,A -85,B 0,C 180,E1 -4884.833,E2 -4884.833} C_VEL
LIN {X 0,Y 523.92,Z 136.848,A -85,B 0,C 180,E1 -4888.002,E2 -4888.002} C_VEL
LIN {X 0,Y 523.927,Z 136.846,A -85,B 0,C 180,E1 -4888.829,E2 -4888.829} C_VEL
LIN {X 0,Y 523.293,Z 136.93,A -85,B 0,C 180,E1 -4889.471,E2 -4889.471} C_VEL
LIN {X 0,Y 520.427,Z 137.286,A -85,B 0,C 180,E1 -4890.513,E2 -4890.513} C_VEL
LIN {X 0,Y 517.991,Z 137.591,A -85,B 0,C 180,E1 -4891.352,E2 -4891.352} C_VEL
LIN {X 0,Y 516.957,Z 137.714,A -85,B 0,C 180,E1 -4892.001,E2 -4892.001} C_VEL
LIN {X 0,Y 516.881,Z 137.722,A -85,B 0,C 180,E1 -4892.22,E2 -4892.22} C_VEL
LIN {X 0,Y 516.886,Z 137.723,A -85,B 0,C 180,E1 -4894.825,E2 -4894.825} C_VEL
LIN {X 0,Y 516.883,Z 137.722,A -85,B 0,C 180,E1 -4897.942,E2 -4897.942} C_VEL
LIN {X 0,Y 516.876,Z 137.721,A -85,B 0,C 180,E1 -4900.743,E2 -4900.743} C_VEL
LIN {X 0,Y 516.886,Z 137.718,A -85,B 0,C 180,E1 -4903.903,E2 -4903.903} C_VEL
LIN {X 0,Y 516.887,Z 137.72,A -85,B 0,C 180,E1 -4906.107,E2 -4906.107} C_VEL
LIN {X 0,Y 516.918,Z 137.718,A -85,B 0,C 180,E1 -4908.398,E2 -4908.398} C_VEL
LIN {X 0,Y 516.882,Z 137.726,A -85,B 0,C 180,E1 -4911.283,E2 -4911.283} C_VEL
LIN {X 0,Y 516.875,Z 137.726,A -85,B 0,C 180,E1 -4914.219,E2 -4914.219} C_VEL
LIN {X 0,Y 516.886,Z 137.727,A -85,B 0,C 180,E1 -4917.052,E2 -4917.052} C_VEL
LIN {X 0,Y 516.891,Z 137.722,A -85,B 0,C 180,E1 -4919.795,E2 -4919.795} C_VEL
LIN {X 0,Y 516.928,Z 137.723,A -85,B 0,C 180,E1 -4922.467,E2 -4922.467} C_VEL
LIN {X 0,Y 516.938,Z 137.779,A -85,B 0,C 180,E1 -4924.965,E2 -4924.965} C_VEL
LIN {X 0,Y 519.219,Z 148.485,A -85,B 0,C 180,E1 -4926.676,E2 -4926.676} C_VEL
LIN {X 0,Y 519.188,Z 159.729,A -85,B 0,C 180,E1 -4928.26,E2 -4928.26} C_VEL
LIN {X 0,Y 522.056,Z 171.929,A -85,B 0,C 180,E1 -4928.576,E2 -4928.576} C_VEL
LIN {X 0,Y 520.994,Z 324.844,A -85,B 0,C 180,E1 -4930.763,E2 -4930.763} C_VEL
LIN {X 0,Y 520.765,Z 340.031,A -85,B 0,C 180,E1 -4931.126,E2 -4931.126} C_VEL
LIN {X 0,Y 520.444,Z 353.813,A -85,B 0,C 180,E1 -4931.599,E2 -4931.599} C_VEL
LIN {X 0,Y 520.113,Z 367.12,A -85,B 0,C 180,E1 -4932.198,E2 -4932.198} C_VEL
LIN {X 0,Y 519.614,Z 381.098,A -85,B 0,C 180,E1 -4932.992,E2 -4932.992} C_VEL
LIN {X 0,Y 519.074,Z 394.196,A -85,B 0,C 180,E1 -4933.914,E2 -4933.914} C_VEL
LIN {X 0,Y 518.573,Z 406.619,A -85,B 0,C 180,E1 -4934.977,E2 -4934.977} C_VEL
LIN {X 0,Y 518.094,Z 417.318,A -85,B 0,C 180,E1 -4936.066,E2 -4936.066} C_VEL
LIN {X 0,Y 517.658,Z 427.16,A -85,B 0,C 180,E1 -4937.254,E2 -4937.254} C_VEL
LIN {X 0,Y 517.25,Z 436.768,A -85,B 0,C 180,E1 -4938.637,E2 -4938.637} C_VEL
LIN {X 0,Y 516.918,Z 444.732,A -85,B 0,C 180,E1 -4940.017,E2 -4940.017} C_VEL
LIN {X 0,Y 516.73,Z 451.316,A -85,B 0,C 180,E1 -4941.395,E2 -4941.395} C_VEL
LIN {X 0,Y 516.541,Z 457.411,A -85,B 0,C 180,E1 -4942.965,E2 -4942.965} C_VEL
LIN {X 0,Y 516.417,Z 462.125,A -85,B 0,C 180,E1 -4944.533,E2 -4944.533} C_VEL
LIN {X 0,Y 516.422,Z 465.576,A -85,B 0,C 180,E1 -4946.097,E2 -4946.097} C_VEL
LIN {X 0,Y 516.273,Z 467.869,A -85,B 0,C 180,E1 -4947.658,E2 -4947.658} C_VEL
LIN {X 0,Y 516.214,Z 469.036,A -85,B 0,C 180,E1 -4949.219,E2 -4949.219} C_VEL
LIN {X 0,Y 516.214,Z 469.053,A -85,B 0,C 180,E1 -4950.779,E2 -4950.779} C_VEL
LIN {X 0,Y 516.273,Z 467.955,A -85,B 0,C 180,E1 -4952.34,E2 -4952.34} C_VEL
LIN {X 0,Y 516.422,Z 465.736,A -85,B 0,C 180,E1 -4953.901,E2 -4953.901} C_VEL
LIN {X 0,Y 516.413,Z 462.367,A -85,B 0,C 180,E1 -4955.466,E2 -4955.466} C_VEL
LIN {X 0,Y 516.539,Z 457.735,A -85,B 0,C 180,E1 -4957.033,E2 -4957.033} C_VEL
LIN {X 0,Y 516.725,Z 451.719,A -85,B 0,C 180,E1 -4958.603,E2 -4958.603} C_VEL
LIN {X 0,Y 516.941,Z 444.152,A -85,B 0,C 180,E1 -4960.179,E2 -4960.179} C_VEL
LIN {X 0,Y 517.277,Z 436.07,A -85,B 0,C 180,E1 -4961.559,E2 -4961.559} C_VEL
LIN {X 0,Y 517.692,Z 426.317,A -85,B 0,C 180,E1 -4962.943,E2 -4962.943} C_VEL
LIN {X 0,Y 518.121,Z 416.351,A -85,B 0,C 180,E1 -4964.131,E2 -4964.131} C_VEL
LIN {X 0,Y 518.645,Z 404.402,A -85,B 0,C 180,E1 -4965.321,E2 -4965.321} C_VEL
LIN {X 0,Y 519.191,Z 392.379,A -85,B 0,C 180,E1 -4966.317,E2 -4966.317} C_VEL
LIN {X 0,Y 519.698,Z 379.403,A -85,B 0,C 180,E1 -4967.206,E2 -4967.206} C_VEL
LIN {X 0,Y 520.151,Z 364.95,A -85,B 0,C 180,E1 -4968.002,E2 -4968.002} C_VEL
LIN {X 0,Y 520.542,Z 351.092,A -85,B 0,C 180,E1 -4968.599,E2 -4968.599} C_VEL
LIN {X 0,Y 520.839,Z 335.384,A -85,B 0,C 180,E1 -4969.096,E2 -4969.096} C_VEL
LIN {X 0,Y 521.057,Z 319.487,A -85,B 0,C 180,E1 -4969.421,E2 -4969.421} C_VEL
LIN {X 0,Y 522.095,Z 172.831,A -85,B 0,C 180,E1 -4971.499,E2 -4971.499} C_VEL
LIN {X 0,Y 519.207,Z 159.808,A -85,B 0,C 180,E1 -4971.82,E2 -4971.82} C_VEL
LIN {X 0,Y 519.296,Z 149.045,A -85,B 0,C 180,E1 -4973.318,E2 -4973.318} C_VEL
LIN {X 0,Y 516.917,Z 137.724,A -85,B 0,C 180,E1 -4975.141,E2 -4975.141} C_VEL
LIN {X 0,Y 516.923,Z 137.722,A -85,B 0,C 180,E1 -4977.904,E2 -4977.904} C_VEL
LIN {X 0,Y 516.889,Z 137.724,A -85,B 0,C 180,E1 -4980.202,E2 -4980.202} C_VEL
LIN {X 0,Y 516.895,Z 137.72,A -85,B 0,C 180,E1 -4982.945,E2 -4982.945} C_VEL
LIN {X 0,Y 516.886,Z 137.725,A -85,B 0,C 180,E1 -4985.778,E2 -4985.778} C_VEL
LIN {X 0,Y 516.877,Z 137.722,A -85,B 0,C 180,E1 -4988.714,E2 -4988.714} C_VEL
LIN {X 0,Y 516.91,Z 137.721,A -85,B 0,C 180,E1 -4991.774,E2 -4991.774} C_VEL
LIN {X 0,Y 516.916,Z 137.718,A -85,B 0,C 180,E1 -4995.009,E2 -4995.009} C_VEL
LIN {X 0,Y 516.915,Z 137.715,A -85,B 0,C 180,E1 -4998.397,E2 -4998.397} C_VEL
LIN {X 0,Y 516.898,Z 137.723,A -85,B 0,C 180,E1 -5001.286,E2 -5001.286} C_VEL
LIN {X 0,Y 516.883,Z 137.72,A -85,B 0,C 180,E1 -5004.22,E2 -5004.22} C_VEL
LIN {X 0,Y 516.889,Z 137.725,A -85,B 0,C 180,E1 -5007.052,E2 -5007.052} C_VEL
LIN {X 0,Y 516.893,Z 137.714,A -85,B 0,C 180,E1 -5009.796,E2 -5009.796} C_VEL
LIN {X 0,Y 516.919,Z 137.717,A -85,B 0,C 180,E1 -5012.467,E2 -5012.467} C_VEL
LIN {X 0,Y 516.901,Z 137.72,A -85,B 0,C 180,E1 -5015.071,E2 -5015.071} C_VEL
LIN {X 0,Y 516.877,Z 137.723,A -85,B 0,C 180,E1 -5018.462,E2 -5018.462} C_VEL
LIN {X 0,Y 516.895,Z 137.72,A -85,B 0,C 180,E1 -5020.954,E2 -5020.954} C_VEL
LIN {X 0,Y 516.907,Z 137.72,A -85,B 0,C 180,E1 -5023.41,E2 -5023.41} C_VEL
LIN {X 0,Y 516.885,Z 137.717,A -85,B 0,C 180,E1 -5025.833,E2 -5025.833} C_VEL
LIN {X 0,Y 516.954,Z 137.708,A -85,B 0,C 180,E1 -5028.233,E2 -5028.233} C_VEL
LIN {X 0,Y 516.96,Z 137.71,A -85,B 0,C 180,E1 -5031.399,E2 -5031.399} C_VEL
LIN {X 0,Y 517,Z 137.699,A -85,B 0,C 180,E1 -5033.757,E2 -5033.757} C_VEL
LIN {X 0,Y 517.007,Z 137.711,A -85,B 0,C 180,E1 -5036.883,E2 -5036.883} C_VEL
LIN {X 0,Y 517.072,Z 137.691,A -85,B 0,C 180,E1 -5040,E2 -5040} C_VEL
LIN {X 0,Y 517.007,Z 137.707,A -85,B 0,C 180,E1 -5043.117,E2 -5043.117} C_VEL
LIN {X 0,Y 516.999,Z 137.705,A -85,B 0,C 180,E1 -5046.243,E2 -5046.243} C_VEL
LIN {X 0,Y 516.948,Z 137.711,A -85,B 0,C 180,E1 -5049.389,E2 -5049.389} C_VEL
LIN {X 0,Y 516.946,Z 137.71,A -85,B 0,C 180,E1 -5051.81,E2 -5051.81} C_VEL
LIN {X 0,Y 516.935,Z 137.713,A -85,B 0,C 180,E1 -5055.148,E2 -5055.148} C_VEL
LIN {X 0,Y 516.915,Z 137.719,A -85,B 0,C 180,E1 -5058.222,E2 -5058.222} C_VEL
LIN {X 0,Y 516.904,Z 137.721,A -85,B 0,C 180,E1 -5060.702,E2 -5060.702} C_VEL
LIN {X 0,Y 516.881,Z 137.718,A -85,B 0,C 180,E1 -5063.223,E2 -5063.223} C_VEL
LIN {X 0,Y 516.932,Z 137.718,A -85,B 0,C 180,E1 -5066.197,E2 -5066.197} C_VEL
LIN {X 0,Y 516.912,Z 137.712,A -85,B 0,C 180,E1 -5069.305,E2 -5069.305} C_VEL
LIN {X 0,Y 516.891,Z 137.723,A -85,B 0,C 180,E1 -5072.545,E2 -5072.545} C_VEL
LIN {X 0,Y 516.873,Z 137.72,A -85,B 0,C 180,E1 -5075.333,E2 -5075.333} C_VEL
LIN {X 0,Y 516.872,Z 137.727,A -85,B 0,C 180,E1 -5077.944,E2 -5077.944} C_VEL
LIN {X 0,Y 516.877,Z 137.713,A -85,B 0,C 180,E1 -5080.742,E2 -5080.742} C_VEL
LIN {X 0,Y 516.876,Z 137.722,A -85,B 0,C 180,E1 -5082.832,E2 -5082.832} C_VEL
LIN {X 0,Y 516.914,Z 137.717,A -85,B 0,C 180,E1 -5085.011,E2 -5085.011} C_VEL
LIN {X 0,Y 516.916,Z 137.721,A -85,B 0,C 180,E1 -5088.398,E2 -5088.398} C_VEL
LIN {X 0,Y 516.879,Z 137.721,A -85,B 0,C 180,E1 -5091.286,E2 -5091.286} C_VEL
LIN {X 0,Y 516.883,Z 137.723,A -85,B 0,C 180,E1 -5094.222,E2 -5094.222} C_VEL
LIN {X 0,Y 516.89,Z 137.72,A -85,B 0,C 180,E1 -5097.054,E2 -5097.054} C_VEL
LIN {X 0,Y 516.895,Z 137.906,A -85,B 0,C 180,E1 -5098.633,E2 -5098.633} C_VEL
LIN {X 0,Y 522.377,Z 156.07,A -85,B 0,C 180,E1 -5100.713,E2 -5100.713} C_VEL
LIN {X 0,Y 521.595,Z 178.439,A -85,B 0,C 180,E1 -5102.784,E2 -5102.784} C_VEL
LIN {X 0,Y 520.393,Z 212.73,A -85,B 0,C 180,E1 -5105.889,E2 -5105.889} C_VEL
LIN {X 0,Y 519.499,Z 241.547,A -85,B 0,C 180,E1 -5108.445,E2 -5108.445} C_VEL
LIN {X 0,Y 521.228,Z 255.204,A -85,B 0,C 180,E1 -5108.717,E2 -5108.717} C_VEL
LIN {X 0,Y 520.137,Z 408.707,A -85,B 0,C 180,E1 -5110.926,E2 -5110.926} C_VEL
LIN {X 0,Y 519.834,Z 424.502,A -85,B 0,C 180,E1 -5111.307,E2 -5111.307} C_VEL
LIN {X 0,Y 519.471,Z 439.411,A -85,B 0,C 180,E1 -5111.827,E2 -5111.827} C_VEL
LIN {X 0,Y 519.029,Z 453.379,A -85,B 0,C 180,E1 -5112.467,E2 -5112.467} C_VEL
LIN {X 0,Y 518.633,Z 467.201,A -85,B 0,C 180,E1 -5113.265,E2 -5113.265} C_VEL
LIN {X 0,Y 518.203,Z 479.908,A -85,B 0,C 180,E1 -5114.162,E2 -5114.162} C_VEL
LIN {X 0,Y 517.728,Z 492.819,A -85,B 0,C 180,E1 -5115.256,E2 -5115.256} C_VEL
LIN {X 0,Y 517.345,Z 504.549,A -85,B 0,C 180,E1 -5116.449,E2 -5116.449} C_VEL
LIN {X 0,Y 517.064,Z 514.411,A -85,B 0,C 180,E1 -5117.64,E2 -5117.64} C_VEL
LIN {X 0,Y 516.839,Z 524.099,A -85,B 0,C 180,E1 -5119.027,E2 -5119.027} C_VEL
LIN {X 0,Y 516.577,Z 532.137,A -85,B 0,C 180,E1 -5120.407,E2 -5120.407} C_VEL
LIN {X 0,Y 516.492,Z 538.811,A -85,B 0,C 180,E1 -5121.787,E2 -5121.787} C_VEL
LIN {X 0,Y 516.413,Z 545.235,A -85,B 0,C 180,E1 -5123.451,E2 -5123.451} C_VEL
LIN {X 0,Y 516.389,Z 548.554,A -85,B 0,C 180,E1 -5124.534,E2 -5124.534} C_VEL
LIN {X 0,Y 516.36,Z 552.227,A -85,B 0,C 180,E1 -5126.099,E2 -5126.099} C_VEL
LIN {X 0,Y 516.291,Z 554.63,A -85,B 0,C 180,E1 -5127.661,E2 -5127.661} C_VEL
LIN {X 0,Y 516.251,Z 555.828,A -85,B 0,C 180,E1 -5129.221,E2 -5129.221} C_VEL
LIN {X 0,Y 516.252,Z 555.812,A -85,B 0,C 180,E1 -5130.781,E2 -5130.781} C_VEL
LIN {X 0,Y 516.295,Z 554.582,A -85,B 0,C 180,E1 -5132.341,E2 -5132.341} C_VEL
LIN {X 0,Y 516.362,Z 552.144,A -85,B 0,C 180,E1 -5133.903,E2 -5133.903} C_VEL
LIN {X 0,Y 516.399,Z 548.433,A -85,B 0,C 180,E1 -5135.468,E2 -5135.468} C_VEL
LIN {X 0,Y 516.459,Z 543.359,A -85,B 0,C 180,E1 -5137.036,E2 -5137.036} C_VEL
LIN {X 0,Y 516.531,Z 536.778,A -85,B 0,C 180,E1 -5138.609,E2 -5138.609} C_VEL
LIN {X 0,Y 516.673,Z 529.675,A -85,B 0,C 180,E1 -5139.988,E2 -5139.988} C_VEL
LIN {X 0,Y 516.863,Z 521.136,A -85,B 0,C 180,E1 -5141.362,E2 -5141.362} C_VEL
LIN {X 0,Y 517.13,Z 510.718,A -85,B 0,C 180,E1 -5142.76,E2 -5142.76} C_VEL
LIN {X 0,Y 517.427,Z 500.086,A -85,B 0,C 180,E1 -5143.952,E2 -5143.952} C_VEL
LIN {X 0,Y 517.847,Z 487.923,A -85,B 0,C 180,E1 -5145.101,E2 -5145.101} C_VEL
LIN {X 0,Y 518.249,Z 474.963,A -85,B 0,C 180,E1 -5146.142,E2 -5146.142} C_VEL
LIN {X 0,Y 518.727,Z 461.429,A -85,B 0,C 180,E1 -5147.038,E2 -5147.038} C_VEL
LIN {X 0,Y 519.187,Z 446.374,A -85,B 0,C 180,E1 -5147.835,E2 -5147.835} C_VEL
LIN {X 0,Y 519.657,Z 430.848,A -85,B 0,C 180,E1 -5148.459,E2 -5148.459} C_VEL
LIN {X 0,Y 519.955,Z 415.855,A -85,B 0,C 180,E1 -5148.897,E2 -5148.897} C_VEL
LIN {X 0,Y 520.157,Z 399.116,A -85,B 0,C 180,E1 -5149.204,E2 -5149.204} C_VEL
LIN {X 0,Y 521.078,Z 255.415,A -85,B 0,C 180,E1 -5151.229,E2 -5151.229} C_VEL
LIN {X 0,Y 519.336,Z 240.568,A -85,B 0,C 180,E1 -5151.536,E2 -5151.536} C_VEL
LIN {X 0,Y 520.228,Z 210.131,A -85,B 0,C 180,E1 -5154.228,E2 -5154.228} C_VEL
LIN {X 0,Y 521.476,Z 176.976,A -85,B 0,C 180,E1 -5157.273,E2 -5157.273} C_VEL
LIN {X 0,Y 522.38,Z 155.894,A -85,B 0,C 180,E1 -5159.3,E2 -5159.3} C_VEL
LIN {X 0,Y 518.656,Z 143.283,A -85,B 0,C 180,E1 -5160.866,E2 -5160.866} C_VEL
LIN {X 0,Y 516.889,Z 137.728,A -85,B 0,C 180,E1 -5161.623,E2 -5161.623} C_VEL
LIN {X 0,Y 516.91,Z 137.726,A -85,B 0,C 180,E1 -5163.966,E2 -5163.966} C_VEL
LIN {X 0,Y 516.855,Z 137.727,A -85,B 0,C 180,E1 -5166.749,E2 -5166.749} C_VEL
LIN {X 0,Y 516.86,Z 137.731,A -85,B 0,C 180,E1 -5169.724,E2 -5169.724} C_VEL
LIN {X 0,Y 516.839,Z 137.73,A -85,B 0,C 180,E1 -5172.837,E2 -5172.837} C_VEL
LIN {X 0,Y 516.899,Z 137.724,A -85,B 0,C 180,E1 -5175.007,E2 -5175.007} C_VEL
LIN {X 0,Y 516.831,Z 137.73,A -85,B 0,C 180,E1 -5178.41,E2 -5178.41} C_VEL
LIN {X 0,Y 516.86,Z 137.731,A -85,B 0,C 180,E1 -5181.282,E2 -5181.282} C_VEL
LIN {X 0,Y 516.852,Z 137.731,A -85,B 0,C 180,E1 -5184.674,E2 -5184.674} C_VEL
LIN {X 0,Y 516.87,Z 137.728,A -85,B 0,C 180,E1 -5187.462,E2 -5187.462} C_VEL
LIN {X 0,Y 516.902,Z 137.726,A -85,B 0,C 180,E1 -5190.694,E2 -5190.694} C_VEL
LIN {X 0,Y 516.879,Z 137.74,A -85,B 0,C 180,E1 -5193.864,E2 -5193.864} C_VEL
LIN {X 0,Y 519.717,Z 149.101,A -85,B 0,C 180,E1 -5196.066,E2 -5196.066} C_VEL
LIN {X 0,Y 520.272,Z 152.68,A -85,B 0,C 180,E1 -5196.719,E2 -5196.719} C_VEL
LIN {X 0,Y 519.535,Z 170.142,A -85,B 0,C 180,E1 -5199.615,E2 -5199.615} C_VEL
LIN {X 0,Y 518.767,Z 190.167,A -85,B 0,C 180,E1 -5202.863,E2 -5202.863} C_VEL
LIN {X 0,Y 518.409,Z 199.252,A -85,B 0,C 180,E1 -5204.318,E2 -5204.318} C_VEL
LIN {X 0,Y 520.086,Z 206.844,A -85,B 0,C 180,E1 -5204.527,E2 -5204.527} C_VEL
LIN {X 0,Y 518.843,Z 311.329,A -85,B 0,C 180,E1 -5206.288,E2 -5206.288} C_VEL
LIN {X 0,Y 518.714,Z 324.949,A -85,B 0,C 180,E1 -5206.684,E2 -5206.684} C_VEL
LIN {X 0,Y 518.576,Z 336.98,A -85,B 0,C 180,E1 -5207.188,E2 -5207.188} C_VEL
LIN {X 0,Y 518.278,Z 349.557,A -85,B 0,C 180,E1 -5207.893,E2 -5207.893} C_VEL
LIN {X 0,Y 518.027,Z 360.232,A -85,B 0,C 180,E1 -5208.655,E2 -5208.655} C_VEL
LIN {X 0,Y 517.781,Z 369.218,A -85,B 0,C 180,E1 -5209.442,E2 -5209.442} C_VEL
LIN {X 0,Y 517.536,Z 378.462,A -85,B 0,C 180,E1 -5210.424,E2 -5210.424} C_VEL
LIN {X 0,Y 517.267,Z 387.364,A -85,B 0,C 180,E1 -5211.602,E2 -5211.602} C_VEL
LIN {X 0,Y 517.02,Z 395.162,A -85,B 0,C 180,E1 -5212.894,E2 -5212.894} C_VEL
LIN {X 0,Y 516.91,Z 401.031,A -85,B 0,C 180,E1 -5214.147,E2 -5214.147} C_VEL
LIN {X 0,Y 516.768,Z 405.314,A -85,B 0,C 180,E1 -5215.32,E2 -5215.32} C_VEL
LIN {X 0,Y 516.694,Z 407.562,A -85,B 0,C 180,E1 -5216.1,E2 -5216.1} C_VEL
LIN {X 0,Y 516.639,Z 409.382,A -85,B 0,C 180,E1 -5216.881,E2 -5216.881} C_VEL
LIN {X 0,Y 516.614,Z 410.758,A -85,B 0,C 180,E1 -5217.661,E2 -5217.661} C_VEL
LIN {X 0,Y 516.634,Z 411.704,A -85,B 0,C 180,E1 -5218.441,E2 -5218.441} C_VEL
LIN {X 0,Y 516.573,Z 412.46,A -85,B 0,C 180,E1 -5220,E2 -5220} C_VEL
LIN {X 0,Y 516.585,Z 412.228,A -85,B 0,C 180,E1 -5220.78,E2 -5220.78} C_VEL
LIN {X 0,Y 516.61,Z 410.572,A -85,B 0,C 180,E1 -5222.339,E2 -5222.339} C_VEL
LIN {X 0,Y 516.583,Z 409.163,A -85,B 0,C 180,E1 -5223.12,E2 -5223.12} C_VEL
LIN {X 0,Y 516.715,Z 406.197,A -85,B 0,C 180,E1 -5224.29,E2 -5224.29} C_VEL
LIN {X 0,Y 516.674,Z 402.234,A -85,B 0,C 180,E1 -5225.464,E2 -5225.464} C_VEL
LIN {X 0,Y 516.889,Z 396.929,A -85,B 0,C 180,E1 -5226.674,E2 -5226.674} C_VEL
LIN {X 0,Y 517.045,Z 390.667,A -85,B 0,C 180,E1 -5227.812,E2 -5227.812} C_VEL
LIN {X 0,Y 517.221,Z 382.63,A -85,B 0,C 180,E1 -5228.99,E2 -5228.99} C_VEL
LIN {X 0,Y 517.436,Z 374.43,A -85,B 0,C 180,E1 -5229.973,E2 -5229.973} C_VEL
LIN {X 0,Y 517.688,Z 364.418,A -85,B 0,C 180,E1 -5230.956,E2 -5230.956} C_VEL
LIN {X 0,Y 517.974,Z 354.55,A -85,B 0,C 180,E1 -5231.743,E2 -5231.743} C_VEL
LIN {X 0,Y 518.204,Z 343.569,A -85,B 0,C 180,E1 -5232.449,E2 -5232.449} C_VEL
LIN {X 0,Y 518.424,Z 331.029,A -85,B 0,C 180,E1 -5233.075,E2 -5233.075} C_VEL
LIN {X 0,Y 518.593,Z 318.984,A -85,B 0,C 180,E1 -5233.519,E2 -5233.519} C_VEL
LIN {X 0,Y 518.733,Z 305.938,A -85,B 0,C 180,E1 -5233.84,E2 -5233.84} C_VEL
LIN {X 0,Y 519.418,Z 205.794,A -85,B 0,C 180,E1 -5235.358,E2 -5235.358} C_VEL
LIN {X 0,Y 517.773,Z 197.079,A -85,B 0,C 180,E1 -5235.553,E2 -5235.553} C_VEL
LIN {X 0,Y 518.269,Z 176.486,A -85,B 0,C 180,E1 -5238.767,E2 -5238.767} C_VEL
LIN {X 0,Y 518.775,Z 159.433,A -85,B 0,C 180,E1 -5241.455,E2 -5241.455} C_VEL
LIN {X 0,Y 519.003,Z 147.698,A -85,B 0,C 180,E1 -5243.334,E2 -5243.334} C_VEL
LIN {X 0,Y 516.934,Z 137.722,A -85,B 0,C 180,E1 -5245.088,E2 -5245.088} C_VEL
LIN {X 0,Y 516.883,Z 137.726,A -85,B 0,C 180,E1 -5247.895,E2 -5247.895} C_VEL
LIN {X 0,Y 516.891,Z 137.721,A -85,B 0,C 180,E1 -5250.204,E2 -5250.204} C_VEL
LIN {X 0,Y 516.881,Z 137.722,A -85,B 0,C 180,E1 -5252.22,E2 -5252.22} C_VEL
LIN {X 0,Y 516.24,Z 137.805,A -85,B 0,C 180,E1 -5252.871,E2 -5252.871} C_VEL
LIN {X 0,Y 513.402,Z 138.162,A -85,B 0,C 180,E1 -5253.927,E2 -5253.927} C_VEL
LIN {X 0,Y 510.976,Z 138.466,A -85,B 0,C 180,E1 -5254.778,E2 -5254.778} C_VEL
LIN {X 0,Y 509.917,Z 138.595,A -85,B 0,C 180,E1 -5255.436,E2 -5255.436} C_VEL
LIN {X 0,Y 509.822,Z 138.605,A -85,B 0,C 180,E1 -5255.658,E2 -5255.658} C_VEL
LIN {X 0,Y 509.853,Z 138.596,A -85,B 0,C 180,E1 -5258.338,E2 -5258.338} C_VEL
LIN {X 0,Y 509.85,Z 138.602,A -85,B 0,C 180,E1 -5261.426,E2 -5261.426} C_VEL
LIN {X 0,Y 509.844,Z 138.598,A -85,B 0,C 180,E1 -5264.67,E2 -5264.67} C_VEL
LIN {X 0,Y 509.837,Z 138.601,A -85,B 0,C 180,E1 -5267.51,E2 -5267.51} C_VEL
LIN {X 0,Y 509.843,Z 138.601,A -85,B 0,C 180,E1 -5270.646,E2 -5270.646} C_VEL
LIN {X 0,Y 509.829,Z 138.602,A -85,B 0,C 180,E1 -5273.646,E2 -5273.646} C_VEL
LIN {X 0,Y 509.846,Z 138.605,A -85,B 0,C 180,E1 -5276.537,E2 -5276.537} C_VEL
LIN {X 0,Y 509.847,Z 138.6,A -85,B 0,C 180,E1 -5279.333,E2 -5279.333} C_VEL
LIN {X 0,Y 509.889,Z 138.596,A -85,B 0,C 180,E1 -5282.053,E2 -5282.053} C_VEL
LIN {X 0,Y 509.885,Z 138.633,A -85,B 0,C 180,E1 -5284.704,E2 -5284.704} C_VEL
LIN {X 0,Y 512.401,Z 150.184,A -85,B 0,C 180,E1 -5286.561,E2 -5286.561} C_VEL
LIN {X 0,Y 512.427,Z 160.143,A -85,B 0,C 180,E1 -5287.958,E2 -5287.958} C_VEL
LIN {X 0,Y 515.45,Z 173.016,A -85,B 0,C 180,E1 -5288.296,E2 -5288.296} C_VEL
LIN {X 0,Y 514.398,Z 316.689,A -85,B 0,C 180,E1 -5290.361,E2 -5290.361} C_VEL
LIN {X 0,Y 514.214,Z 332.385,A -85,B 0,C 180,E1 -5290.653,E2 -5290.653} C_VEL
LIN {X 0,Y 513.941,Z 347.598,A -85,B 0,C 180,E1 -5291.099,E2 -5291.099} C_VEL
LIN {X 0,Y 513.55,Z 362.475,A -85,B 0,C 180,E1 -5291.705,E2 -5291.705} C_VEL
LIN {X 0,Y 513.054,Z 376.746,A -85,B 0,C 180,E1 -5292.46,E2 -5292.46} C_VEL
LIN {X 0,Y 512.461,Z 390.395,A -85,B 0,C 180,E1 -5293.364,E2 -5293.364} C_VEL
LIN {X 0,Y 511.926,Z 402.799,A -85,B 0,C 180,E1 -5294.369,E2 -5294.369} C_VEL
LIN {X 0,Y 511.371,Z 414.179,A -85,B 0,C 180,E1 -5295.473,E2 -5295.473} C_VEL
LIN {X 0,Y 510.921,Z 424.6,A -85,B 0,C 180,E1 -5296.678,E2 -5296.678} C_VEL
LIN {X 0,Y 510.38,Z 434.744,A -85,B 0,C 180,E1 -5298.079,E2 -5298.079} C_VEL
LIN {X 0,Y 510.095,Z 443.158,A -85,B 0,C 180,E1 -5299.48,E2 -5299.48} C_VEL
LIN {X 0,Y 509.798,Z 450.159,A -85,B 0,C 180,E1 -5300.877,E2 -5300.877} C_VEL
LIN {X 0,Y 509.544,Z 456.628,A -85,B 0,C 180,E1 -5302.47,E2 -5302.47} C_VEL
LIN {X 0,Y 509.432,Z 461.683,A -85,B 0,C 180,E1 -5304.06,E2 -5304.06} C_VEL
LIN {X 0,Y 509.339,Z 464.589,A -85,B 0,C 180,E1 -5305.25,E2 -5305.25} C_VEL
LIN {X 0,Y 509.301,Z 467.448,A -85,B 0,C 180,E1 -5306.835,E2 -5306.835} C_VEL
LIN {X 0,Y 509.153,Z 469.176,A -85,B 0,C 180,E1 -5308.417,E2 -5308.417} C_VEL
LIN {X 0,Y 509.135,Z 469.774,A -85,B 0,C 180,E1 -5309.999,E2 -5309.999} C_VEL
LIN {X 0,Y 509.151,Z 469.227,A -85,B 0,C 180,E1 -5311.581,E2 -5311.581} C_VEL
LIN {X 0,Y 509.302,Z 467.569,A -85,B 0,C 180,E1 -5313.163,E2 -5313.163} C_VEL
LIN {X 0,Y 509.338,Z 464.786,A -85,B 0,C 180,E1 -5314.748,E2 -5314.748} C_VEL
LIN {X 0,Y 509.43,Z 460.797,A -85,B 0,C 180,E1 -5316.335,E2 -5316.335} C_VEL
LIN {X 0,Y 509.564,Z 455.493,A -85,B 0,C 180,E1 -5317.927,E2 -5317.927} C_VEL
LIN {X 0,Y 509.847,Z 448.72,A -85,B 0,C 180,E1 -5319.52,E2 -5319.52} C_VEL
LIN {X 0,Y 510.171,Z 441.463,A -85,B 0,C 180,E1 -5320.918,E2 -5320.918} C_VEL
LIN {X 0,Y 510.539,Z 431.791,A -85,B 0,C 180,E1 -5322.449,E2 -5322.449} C_VEL
LIN {X 0,Y 511.044,Z 422.112,A -85,B 0,C 180,E1 -5323.722,E2 -5323.722} C_VEL
LIN {X 0,Y 511.548,Z 411.222,A -85,B 0,C 180,E1 -5324.927,E2 -5324.927} C_VEL
LIN {X 0,Y 512.095,Z 399.159,A -85,B 0,C 180,E1 -5326.04,E2 -5326.04} C_VEL
LIN {X 0,Y 512.691,Z 386.052,A -85,B 0,C 180,E1 -5327.037,E2 -5327.037} C_VEL
LIN {X 0,Y 513.215,Z 373.149,A -85,B 0,C 180,E1 -5327.841,E2 -5327.841} C_VEL
LIN {X 0,Y 513.644,Z 359.001,A -85,B 0,C 180,E1 -5328.548,E2 -5328.548} C_VEL
LIN {X 0,Y 514.042,Z 344.409,A -85,B 0,C 180,E1 -5329.102,E2 -5329.102} C_VEL
LIN {X 0,Y 514.261,Z 329.636,A -85,B 0,C 180,E1 -5329.503,E2 -5329.503} C_VEL
LIN {X 0,Y 514.479,Z 308.542,A -85,B 0,C 180,E1 -5329.845,E2 -5329.845} C_VEL
LIN {X 0,Y 515.421,Z 172.914,A -85,B 0,C 180,E1 -5331.797,E2 -5331.797} C_VEL
LIN {X 0,Y 512.428,Z 160.108,A -85,B 0,C 180,E1 -5332.139,E2 -5332.139} C_VEL
LIN {X 0,Y 512.479,Z 150.758,A -85,B 0,C 180,E1 -5333.433,E2 -5333.433} C_VEL
LIN {X 0,Y 509.88,Z 138.601,A -85,B 0,C 180,E1 -5335.404,E2 -5335.404} C_VEL
LIN {X 0,Y 509.895,Z 138.595,A -85,B 0,C 180,E1 -5338.1,E2 -5338.1} C_VEL
LIN {X 0,Y 509.844,Z 138.604,A -85,B 0,C 180,E1 -5341.279,E2 -5341.279} C_VEL
LIN {X 0,Y 509.857,Z 138.598,A -85,B 0,C 180,E1 -5344.202,E2 -5344.202} C_VEL
LIN {X 0,Y 509.814,Z 138.607,A -85,B 0,C 180,E1 -5347.339,E2 -5347.339} C_VEL
LIN {X 0,Y 509.833,Z 138.59,A -85,B 0,C 180,E1 -5350.381,E2 -5350.381} C_VEL
LIN {X 0,Y 509.834,Z 138.604,A -85,B 0,C 180,E1 -5353.063,E2 -5353.063} C_VEL
LIN {X 0,Y 509.824,Z 138.603,A -85,B 0,C 180,E1 -5355.791,E2 -5355.791} C_VEL
LIN {X 0,Y 509.858,Z 138.595,A -85,B 0,C 180,E1 -5358.575,E2 -5358.575} C_VEL
LIN {X 0,Y 509.851,Z 138.598,A -85,B 0,C 180,E1 -5361.662,E2 -5361.662} C_VEL
LIN {X 0,Y 509.838,Z 138.599,A -85,B 0,C 180,E1 -5364.622,E2 -5364.622} C_VEL
LIN {X 0,Y 509.857,Z 138.6,A -85,B 0,C 180,E1 -5367.48,E2 -5367.48} C_VEL
LIN {X 0,Y 509.872,Z 138.588,A -85,B 0,C 180,E1 -5370.268,E2 -5370.268} C_VEL
LIN {X 0,Y 509.876,Z 138.6,A -85,B 0,C 180,E1 -5372.944,E2 -5372.944} C_VEL
LIN {X 0,Y 509.86,Z 138.594,A -85,B 0,C 180,E1 -5375.573,E2 -5375.573} C_VEL
LIN {X 0,Y 509.812,Z 138.601,A -85,B 0,C 180,E1 -5378.148,E2 -5378.148} C_VEL
LIN {X 0,Y 509.855,Z 138.597,A -85,B 0,C 180,E1 -5380.681,E2 -5380.681} C_VEL
LIN {X 0,Y 509.877,Z 138.598,A -85,B 0,C 180,E1 -5383.174,E2 -5383.174} C_VEL
LIN {X 0,Y 509.854,Z 138.593,A -85,B 0,C 180,E1 -5385.634,E2 -5385.634} C_VEL
LIN {X 0,Y 509.907,Z 138.594,A -85,B 0,C 180,E1 -5388.874,E2 -5388.874} C_VEL
LIN {X 0,Y 509.941,Z 138.584,A -85,B 0,C 180,E1 -5392.078,E2 -5392.078} C_VEL
LIN {X 0,Y 509.973,Z 138.578,A -85,B 0,C 180,E1 -5394.464,E2 -5394.464} C_VEL
LIN {X 0,Y 510.044,Z 138.572,A -85,B 0,C 180,E1 -5397.631,E2 -5397.631} C_VEL
LIN {X 0,Y 510.056,Z 138.571,A -85,B 0,C 180,E1 -5400.789,E2 -5400.789} C_VEL
LIN {X 0,Y 509.949,Z 138.586,A -85,B 0,C 180,E1 -5403.16,E2 -5403.16} C_VEL
LIN {X 0,Y 509.967,Z 138.582,A -85,B 0,C 180,E1 -5406.33,E2 -5406.33} C_VEL
LIN {X 0,Y 509.908,Z 138.594,A -85,B 0,C 180,E1 -5408.72,E2 -5408.72} C_VEL
LIN {X 0,Y 509.894,Z 138.589,A -85,B 0,C 180,E1 -5411.932,E2 -5411.932} C_VEL
LIN {X 0,Y 509.882,Z 138.591,A -85,B 0,C 180,E1 -5415.242,E2 -5415.242} C_VEL
LIN {X 0,Y 509.878,Z 138.593,A -85,B 0,C 180,E1 -5418.001,E2 -5418.001} C_VEL
LIN {X 0,Y 509.847,Z 138.597,A -85,B 0,C 180,E1 -5421.002,E2 -5421.002} C_VEL
LIN {X 0,Y 509.84,Z 138.595,A -85,B 0,C 180,E1 -5423.563,E2 -5423.563} C_VEL
LIN {X 0,Y 509.901,Z 138.597,A -85,B 0,C 180,E1 -5426.379,E2 -5426.379} C_VEL
LIN {X 0,Y 509.867,Z 138.592,A -85,B 0,C 180,E1 -5428.845,E2 -5428.845} C_VEL
LIN {X 0,Y 509.815,Z 138.601,A -85,B 0,C 180,E1 -5431.59,E2 -5431.59} C_VEL
LIN {X 0,Y 509.844,Z 138.601,A -85,B 0,C 180,E1 -5434.414,E2 -5434.414} C_VEL
LIN {X 0,Y 509.81,Z 138.601,A -85,B 0,C 180,E1 -5437.341,E2 -5437.341} C_VEL
LIN {X 0,Y 509.829,Z 138.589,A -85,B 0,C 180,E1 -5440.383,E2 -5440.383} C_VEL
LIN {X 0,Y 509.815,Z 138.6,A -85,B 0,C 180,E1 -5443.063,E2 -5443.063} C_VEL
LIN {X 0,Y 509.823,Z 138.605,A -85,B 0,C 180,E1 -5445.793,E2 -5445.793} C_VEL
LIN {X 0,Y 509.858,Z 138.598,A -85,B 0,C 180,E1 -5448.577,E2 -5448.577} C_VEL
LIN {X 0,Y 509.845,Z 138.602,A -85,B 0,C 180,E1 -5451.787,E2 -5451.787} C_VEL
LIN {X 0,Y 509.837,Z 138.597,A -85,B 0,C 180,E1 -5454.624,E2 -5454.624} C_VEL
LIN {X 0,Y 509.857,Z 138.599,A -85,B 0,C 180,E1 -5457.482,E2 -5457.482} C_VEL
LIN {X 0,Y 509.854,Z 138.714,A -85,B 0,C 180,E1 -5458.283,E2 -5458.283} C_VEL
LIN {X 0,Y 515.632,Z 157.879,A -85,B 0,C 180,E1 -5460.516,E2 -5460.516} C_VEL
LIN {X 0,Y 515.529,Z 164.205,A -85,B 0,C 180,E1 -5461.122,E2 -5461.122} C_VEL
LIN {X 0,Y 514.178,Z 197.421,A -85,B 0,C 180,E1 -5464.207,E2 -5464.207} C_VEL
LIN {X 0,Y 513.071,Z 228.367,A -85,B 0,C 180,E1 -5467.023,E2 -5467.023} C_VEL
LIN {X 0,Y 512.654,Z 241.298,A -85,B 0,C 180,E1 -5468.184,E2 -5468.184} C_VEL
LIN {X 0,Y 514.498,Z 257.256,A -85,B 0,C 180,E1 -5468.499,E2 -5468.499} C_VEL
LIN {X 0,Y 513.356,Z 408.223,A -85,B 0,C 180,E1 -5470.69,E2 -5470.69} C_VEL
LIN {X 0,Y 513.033,Z 423.701,A -85,B 0,C 180,E1 -5471.069,E2 -5471.069} C_VEL
LIN {X 0,Y 512.605,Z 439.073,A -85,B 0,C 180,E1 -5471.62,E2 -5471.62} C_VEL
LIN {X 0,Y 512.074,Z 453.815,A -85,B 0,C 180,E1 -5472.324,E2 -5472.324} C_VEL
LIN {X 0,Y 511.604,Z 468.8,A -85,B 0,C 180,E1 -5473.234,E2 -5473.234} C_VEL
LIN {X 0,Y 511.141,Z 481.441,A -85,B 0,C 180,E1 -5474.166,E2 -5474.166} C_VEL
LIN {X 0,Y 510.656,Z 493.719,A -85,B 0,C 180,E1 -5475.251,E2 -5475.251} C_VEL
LIN {X 0,Y 510.266,Z 505.179,A -85,B 0,C 180,E1 -5476.46,E2 -5476.46} C_VEL
LIN {X 0,Y 509.982,Z 514.839,A -85,B 0,C 180,E1 -5477.668,E2 -5477.668} C_VEL
LIN {X 0,Y 509.729,Z 524.306,A -85,B 0,C 180,E1 -5479.073,E2 -5479.073} C_VEL
LIN {X 0,Y 509.477,Z 532.151,A -85,B 0,C 180,E1 -5480.473,E2 -5480.473} C_VEL
LIN {X 0,Y 509.397,Z 539.483,A -85,B 0,C 180,E1 -5482.071,E2 -5482.071} C_VEL
LIN {X 0,Y 509.383,Z 545.247,A -85,B 0,C 180,E1 -5483.664,E2 -5483.664} C_VEL
LIN {X 0,Y 509.283,Z 549.586,A -85,B 0,C 180,E1 -5485.252,E2 -5485.252} C_VEL
LIN {X 0,Y 509.29,Z 552.632,A -85,B 0,C 180,E1 -5486.837,E2 -5486.837} C_VEL
LIN {X 0,Y 509.205,Z 554.423,A -85,B 0,C 180,E1 -5488.419,E2 -5488.419} C_VEL
LIN {X 0,Y 509.23,Z 555.023,A -85,B 0,C 180,E1 -5490.001,E2 -5490.001} C_VEL
LIN {X 0,Y 509.212,Z 554.368,A -85,B 0,C 180,E1 -5491.583,E2 -5491.583} C_VEL
LIN {X 0,Y 509.3,Z 552.522,A -85,B 0,C 180,E1 -5493.165,E2 -5493.165} C_VEL
LIN {X 0,Y 509.302,Z 549.422,A -85,B 0,C 180,E1 -5494.75,E2 -5494.75} C_VEL
LIN {X 0,Y 509.365,Z 545.011,A -85,B 0,C 180,E1 -5496.338,E2 -5496.338} C_VEL
LIN {X 0,Y 509.43,Z 539.157,A -85,B 0,C 180,E1 -5497.931,E2 -5497.931} C_VEL
LIN {X 0,Y 509.497,Z 531.696,A -85,B 0,C 180,E1 -5499.529,E2 -5499.529} C_VEL
LIN {X 0,Y 509.731,Z 523.725,A -85,B 0,C 180,E1 -5500.929,E2 -5500.929} C_VEL
LIN {X 0,Y 509.982,Z 514.122,A -85,B 0,C 180,E1 -5502.335,E2 -5502.335} C_VEL
LIN {X 0,Y 510.262,Z 504.595,A -85,B 0,C 180,E1 -5503.542,E2 -5503.542} C_VEL
LIN {X 0,Y 510.69,Z 492.234,A -85,B 0,C 180,E1 -5504.852,E2 -5504.852} C_VEL
LIN {X 0,Y 511.195,Z 479.617,A -85,B 0,C 180,E1 -5505.961,E2 -5505.961} C_VEL
LIN {X 0,Y 511.631,Z 467.233,A -85,B 0,C 180,E1 -5506.87,E2 -5506.87} C_VEL
LIN {X 0,Y 512.127,Z 453.811,A -85,B 0,C 180,E1 -5507.676,E2 -5507.676} C_VEL
LIN {X 0,Y 512.675,Z 439.025,A -85,B 0,C 180,E1 -5508.38,E2 -5508.38} C_VEL
LIN {X 0,Y 513.03,Z 424.045,A -85,B 0,C 180,E1 -5508.919,E2 -5508.919} C_VEL
LIN {X 0,Y 513.345,Z 409.356,A -85,B 0,C 180,E1 -5509.287,E2 -5509.287} C_VEL
LIN {X 0,Y 513.769,Z 357.476,A -85,B 0,C 180,E1 -5510.051,E2 -5510.051} C_VEL
LIN {X 0,Y 514.322,Z 254.737,A -85,B 0,C 180,E1 -5511.524,E2 -5511.524} C_VEL
LIN {X 0,Y 512.498,Z 239.744,A -85,B 0,C 180,E1 -5511.838,E2 -5511.838} C_VEL
LIN {X 0,Y 513.553,Z 207.235,A -85,B 0,C 180,E1 -5514.779,E2 -5514.779} C_VEL
LIN {X 0,Y 514.876,Z 176.768,A -85,B 0,C 180,E1 -5517.653,E2 -5517.653} C_VEL
LIN {X 0,Y 515.861,Z 159.23,A -85,B 0,C 180,E1 -5519.372,E2 -5519.372} C_VEL
LIN {X 0,Y 514.725,Z 154.061,A -85,B 0,C 180,E1 -5519.99,E2 -5519.99} C_VEL
LIN {X 0,Y 511.09,Z 142.638,A -85,B 0,C 180,E1 -5521.509,E2 -5521.509} C_VEL
LIN {X 0,Y 509.849,Z 138.604,A -85,B 0,C 180,E1 -5522.082,E2 -5522.082} C_VEL
LIN {X 0,Y 509.849,Z 138.604,A -85,B 0,C 180,E1 -5524.414,E2 -5524.414} C_VEL
LIN {X 0,Y 509.809,Z 138.609,A -85,B 0,C 180,E1 -5527.342,E2 -5527.342} C_VEL
LIN {X 0,Y 509.814,Z 138.605,A -85,B 0,C 180,E1 -5530.385,E2 -5530.385} C_VEL
LIN {X 0,Y 509.793,Z 138.611,A -85,B 0,C 180,E1 -5533.576,E2 -5533.576} C_VEL
LIN {X 0,Y 509.794,Z 138.606,A -85,B 0,C 180,E1 -5536.426,E2 -5536.426} C_VEL
LIN {X 0,Y 509.788,Z 138.61,A -85,B 0,C 180,E1 -5539.613,E2 -5539.613} C_VEL
LIN {X 0,Y 509.776,Z 138.612,A -85,B 0,C 180,E1 -5542.656,E2 -5542.656} C_VEL
LIN {X 0,Y 509.841,Z 138.602,A -85,B 0,C 180,E1 -5545.801,E2 -5545.801} C_VEL
LIN {X 0,Y 509.818,Z 138.609,A -85,B 0,C 180,E1 -5548.726,E2 -5548.726} C_VEL
LIN {X 0,Y 509.837,Z 138.606,A -85,B 0,C 180,E1 -5551.153,E2 -5551.153} C_VEL
LIN {X 0,Y 509.854,Z 138.754,A -85,B 0,C 180,E1 -5553.432,E2 -5553.432} C_VEL
LIN {X 0,Y 512.826,Z 150.231,A -85,B 0,C 180,E1 -5555.724,E2 -5555.724} C_VEL
LIN {X 0,Y 513.621,Z 155.001,A -85,B 0,C 180,E1 -5556.621,E2 -5556.621} C_VEL
LIN {X 0,Y 512.789,Z 172.416,A -85,B 0,C 180,E1 -5559.544,E2 -5559.544} C_VEL
LIN {X 0,Y 511.936,Z 192.401,A -85,B 0,C 180,E1 -5562.833,E2 -5562.833} C_VEL
LIN {X 0,Y 511.682,Z 200.069,A -85,B 0,C 180,E1 -5564.042,E2 -5564.042} C_VEL
LIN {X 0,Y 513.444,Z 208.056,A -85,B 0,C 180,E1 -5564.269,E2 -5564.269} C_VEL
LIN {X 0,Y 511.996,Z 312.591,A -85,B 0,C 180,E1 -5566.101,E2 -5566.101} C_VEL
LIN {X 0,Y 511.869,Z 326.001,A -85,B 0,C 180,E1 -5566.502,E2 -5566.502} C_VEL
LIN {X 0,Y 511.723,Z 337.954,A -85,B 0,C 180,E1 -5567.014,E2 -5567.014} C_VEL
LIN {X 0,Y 511.39,Z 350.629,A -85,B 0,C 180,E1 -5567.736,E2 -5567.736} C_VEL
LIN {X 0,Y 511.146,Z 361.169,A -85,B 0,C 180,E1 -5568.5,E2 -5568.5} C_VEL
LIN {X 0,Y 510.842,Z 371.207,A -85,B 0,C 180,E1 -5569.397,E2 -5569.397} C_VEL
LIN {X 0,Y 510.589,Z 381.03,A -85,B 0,C 180,E1 -5570.493,E2 -5570.493} C_VEL
LIN {X 0,Y 510.291,Z 389.675,A -85,B 0,C 180,E1 -5571.685,E2 -5571.685} C_VEL
LIN {X 0,Y 509.997,Z 396.573,A -85,B 0,C 180,E1 -5572.876,E2 -5572.876} C_VEL
LIN {X 0,Y 509.929,Z 402.038,A -85,B 0,C 180,E1 -5574.067,E2 -5574.067} C_VEL
LIN {X 0,Y 509.766,Z 406.33,A -85,B 0,C 180,E1 -5575.255,E2 -5575.255} C_VEL
LIN {X 0,Y 509.683,Z 408.578,A -85,B 0,C 180,E1 -5576.047,E2 -5576.047} C_VEL
LIN {X 0,Y 509.623,Z 410.399,A -85,B 0,C 180,E1 -5576.838,E2 -5576.838} C_VEL
LIN {X 0,Y 509.602,Z 411.774,A -85,B 0,C 180,E1 -5577.629,E2 -5577.629} C_VEL
LIN {X 0,Y 509.626,Z 412.715,A -85,B 0,C 180,E1 -5578.42,E2 -5578.42} C_VEL
LIN {X 0,Y 509.556,Z 413.454,A -85,B 0,C 180,E1 -5580,E2 -5580} C_VEL
LIN {X 0,Y 509.569,Z 413.212,A -85,B 0,C 180,E1 -5580.79,E2 -5580.79} C_VEL
LIN {X 0,Y 509.51,Z 412.574,A -85,B 0,C 180,E1 -5581.581,E2 -5581.581} C_VEL
LIN {X 0,Y 509.595,Z 411.526,A -85,B 0,C 180,E1 -5582.371,E2 -5582.371} C_VEL
LIN {X 0,Y 509.556,Z 410.101,A -85,B 0,C 180,E1 -5583.163,E2 -5583.163} C_VEL
LIN {X 0,Y 509.698,Z 407.105,A -85,B 0,C 180,E1 -5584.349,E2 -5584.349} C_VEL
LIN {X 0,Y 509.671,Z 403.107,A -85,B 0,C 180,E1 -5585.539,E2 -5585.539} C_VEL
LIN {X 0,Y 509.898,Z 397.819,A -85,B 0,C 180,E1 -5586.755,E2 -5586.755} C_VEL
LIN {X 0,Y 510.061,Z 391.461,A -85,B 0,C 180,E1 -5587.92,E2 -5587.92} C_VEL
LIN {X 0,Y 510.259,Z 383.379,A -85,B 0,C 180,E1 -5589.114,E2 -5589.114} C_VEL
LIN {X 0,Y 510.496,Z 375.13,A -85,B 0,C 180,E1 -5590.11,E2 -5590.11} C_VEL
LIN {X 0,Y 510.768,Z 365.07,A -85,B 0,C 180,E1 -5591.107,E2 -5591.107} C_VEL
LIN {X 0,Y 511.062,Z 355.15,A -85,B 0,C 180,E1 -5591.904,E2 -5591.904} C_VEL
LIN {X 0,Y 511.292,Z 344.593,A -85,B 0,C 180,E1 -5592.593,E2 -5592.593} C_VEL
LIN {X 0,Y 511.543,Z 331.526,A -85,B 0,C 180,E1 -5593.254,E2 -5593.254} C_VEL
LIN {X 0,Y 511.727,Z 319.435,A -85,B 0,C 180,E1 -5593.704,E2 -5593.704} C_VEL
LIN {X 0,Y 511.867,Z 306.273,A -85,B 0,C 180,E1 -5594.03,E2 -5594.03} C_VEL
LIN {X 0,Y 512.558,Z 206.296,A -85,B 0,C 180,E1 -5595.582,E2 -5595.582} C_VEL
LIN {X 0,Y 510.827,Z 197.271,A -85,B 0,C 180,E1 -5595.796,E2 -5595.796} C_VEL
LIN {X 0,Y 511.396,Z 176.622,A -85,B 0,C 180,E1 -5599.05,E2 -5599.05} C_VEL
LIN {X 0,Y 511.942,Z 158.313,A -85,B 0,C 180,E1 -5601.968,E2 -5601.968} C_VEL
LIN {X 0,Y 512.12,Z 149.156,A -85,B 0,C 180,E1 -5603.452,E2 -5603.452} C_VEL
LIN {X 0,Y 509.854,Z 138.604,A -85,B 0,C 180,E1 -5605.325,E2 -5605.325} C_VEL
LIN {X 0,Y 509.835,Z 138.602,A -85,B 0,C 180,E1 -5608.086,E2 -5608.086} C_VEL
LIN {X 0,Y 509.847,Z 138.599,A -85,B 0,C 180,E1 -5610.666,E2 -5610.666} C_VEL
LIN {X 0,Y 509.863,Z 138.603,A -85,B 0,C 180,E1 -5613.461,E2 -5613.461} C_VEL
LIN {X 0,Y 509.822,Z 138.605,A -85,B 0,C 180,E1 -5615.658,E2 -5615.658} C_VEL
LIN {X 0,Y 509.14,Z 138.686,A -85,B 0,C 180,E1 -5616.318,E2 -5616.318} C_VEL
LIN {X 0,Y 506.308,Z 139.045,A -85,B 0,C 180,E1 -5617.39,E2 -5617.39} C_VEL
LIN {X 0,Y 503.919,Z 139.345,A -85,B 0,C 180,E1 -5618.253,E2 -5618.253} C_VEL
LIN {X 0,Y 502.883,Z 139.47,A -85,B 0,C 180,E1 -5618.919,E2 -5618.919} C_VEL
LIN {X 0,Y 502.792,Z 139.479,A -85,B 0,C 180,E1 -5619.145,E2 -5619.145} C_VEL
LIN {X 0,Y 502.808,Z 139.475,A -85,B 0,C 180,E1 -5622.199,E2 -5622.199} C_VEL
LIN {X 0,Y 502.791,Z 139.48,A -85,B 0,C 180,E1 -5625.47,E2 -5625.47} C_VEL
LIN {X 0,Y 502.824,Z 139.48,A -85,B 0,C 180,E1 -5628.934,E2 -5628.934} C_VEL
LIN {X 0,Y 502.797,Z 139.478,A -85,B 0,C 180,E1 -5632.046,E2 -5632.046} C_VEL
LIN {X 0,Y 502.8,Z 139.482,A -85,B 0,C 180,E1 -5635.033,E2 -5635.033} C_VEL
LIN {X 0,Y 502.787,Z 139.479,A -85,B 0,C 180,E1 -5637.915,E2 -5637.915} C_VEL
LIN {X 0,Y 502.826,Z 139.48,A -85,B 0,C 180,E1 -5640.711,E2 -5640.711} C_VEL
LIN {X 0,Y 502.868,Z 139.471,A -85,B 0,C 180,E1 -5643.439,E2 -5643.439} C_VEL
LIN {X 0,Y 502.859,Z 139.491,A -85,B 0,C 180,E1 -5644.434,E2 -5644.434} C_VEL
LIN {X 0,Y 505.485,Z 151.484,A -85,B 0,C 180,E1 -5646.375,E2 -5646.375} C_VEL
LIN {X 0,Y 505.699,Z 156.55,A -85,B 0,C 180,E1 -5647.099,E2 -5647.099} C_VEL
LIN {X 0,Y 505.644,Z 160.627,A -85,B 0,C 180,E1 -5647.651,E2 -5647.651} C_VEL
LIN {X 0,Y 508.898,Z 174.933,A -85,B 0,C 180,E1 -5648.024,E2 -5648.024} C_VEL
LIN {X 0,Y 507.644,Z 325.577,A -85,B 0,C 180,E1 -5650.232,E2 -5650.232} C_VEL
LIN {X 0,Y 507.423,Z 340.214,A -85,B 0,C 180,E1 -5650.584,E2 -5650.584} C_VEL
LIN {X 0,Y 507.103,Z 353.659,A -85,B 0,C 180,E1 -5651.044,E2 -5651.044} C_VEL
LIN {X 0,Y 506.736,Z 366.247,A -85,B 0,C 180,E1 -5651.607,E2 -5651.607} C_VEL
LIN {X 0,Y 506.157,Z 380.682,A -85,B 0,C 180,E1 -5652.421,E2 -5652.421} C_VEL
LIN {X 0,Y 505.577,Z 393.701,A -85,B 0,C 180,E1 -5653.339,E2 -5653.339} C_VEL
LIN {X 0,Y 505.002,Z 405.672,A -85,B 0,C 180,E1 -5654.36,E2 -5654.36} C_VEL
LIN {X 0,Y 504.421,Z 416.636,A -85,B 0,C 180,E1 -5655.475,E2 -5655.475} C_VEL
LIN {X 0,Y 503.927,Z 426.749,A -85,B 0,C 180,E1 -5656.695,E2 -5656.695} C_VEL
LIN {X 0,Y 503.409,Z 436.629,A -85,B 0,C 180,E1 -5658.116,E2 -5658.116} C_VEL
LIN {X 0,Y 503.01,Z 444.823,A -85,B 0,C 180,E1 -5659.534,E2 -5659.534} C_VEL
LIN {X 0,Y 502.738,Z 452.484,A -85,B 0,C 180,E1 -5661.153,E2 -5661.153} C_VEL
LIN {X 0,Y 502.492,Z 458.58,A -85,B 0,C 180,E1 -5662.768,E2 -5662.768} C_VEL
LIN {X 0,Y 502.313,Z 463.296,A -85,B 0,C 180,E1 -5664.379,E2 -5664.379} C_VEL
LIN {X 0,Y 502.305,Z 466.746,A -85,B 0,C 180,E1 -5665.987,E2 -5665.987} C_VEL
LIN {X 0,Y 502.137,Z 469.039,A -85,B 0,C 180,E1 -5667.593,E2 -5667.593} C_VEL
LIN {X 0,Y 502.064,Z 470.205,A -85,B 0,C 180,E1 -5669.197,E2 -5669.197} C_VEL
LIN {X 0,Y 502.064,Z 470.223,A -85,B 0,C 180,E1 -5670.801,E2 -5670.801} C_VEL
LIN {X 0,Y 502.137,Z 469.122,A -85,B 0,C 180,E1 -5672.405,E2 -5672.405} C_VEL
LIN {X 0,Y 502.29,Z 466.903,A -85,B 0,C 180,E1 -5674.011,E2 -5674.011} C_VEL
LIN {X 0,Y 502.306,Z 463.532,A -85,B 0,C 180,E1 -5675.619,E2 -5675.619} C_VEL
LIN {X 0,Y 502.48,Z 458.897,A -85,B 0,C 180,E1 -5677.23,E2 -5677.23} C_VEL
LIN {X 0,Y 502.733,Z 452.876,A -85,B 0,C 180,E1 -5678.845,E2 -5678.845} C_VEL
LIN {X 0,Y 502.992,Z 445.305,A -85,B 0,C 180,E1 -5680.464,E2 -5680.464} C_VEL
LIN {X 0,Y 503.404,Z 437.216,A -85,B 0,C 180,E1 -5681.882,E2 -5681.882} C_VEL
LIN {X 0,Y 503.869,Z 427.457,A -85,B 0,C 180,E1 -5683.304,E2 -5683.304} C_VEL
LIN {X 0,Y 504.391,Z 417.479,A -85,B 0,C 180,E1 -5684.524,E2 -5684.524} C_VEL
LIN {X 0,Y 505.002,Z 405.553,A -85,B 0,C 180,E1 -5685.742,E2 -5685.742} C_VEL
LIN {X 0,Y 505.603,Z 393.817,A -85,B 0,C 180,E1 -5686.742,E2 -5686.742} C_VEL
LIN {X 0,Y 506.189,Z 380.483,A -85,B 0,C 180,E1 -5687.68,E2 -5687.68} C_VEL
LIN {X 0,Y 506.707,Z 365.997,A -85,B 0,C 180,E1 -5688.497,E2 -5688.497} C_VEL
LIN {X 0,Y 507.181,Z 351.381,A -85,B 0,C 180,E1 -5689.134,E2 -5689.134} C_VEL
LIN {X 0,Y 507.493,Z 336.019,A -85,B 0,C 180,E1 -5689.625,E2 -5689.625} C_VEL
LIN {X 0,Y 507.729,Z 320.343,A -85,B 0,C 180,E1 -5689.949,E2 -5689.949} C_VEL
LIN {X 0,Y 508.928,Z 174.946,A -85,B 0,C 180,E1 -5692.065,E2 -5692.065} C_VEL
LIN {X 0,Y 505.689,Z 160.553,A -85,B 0,C 180,E1 -5692.45,E2 -5692.45} C_VEL
LIN {X 0,Y 505.634,Z 152.067,A -85,B 0,C 180,E1 -5693.623,E2 -5693.623} C_VEL
LIN {X 0,Y 502.861,Z 139.476,A -85,B 0,C 180,E1 -5695.673,E2 -5695.673} C_VEL
LIN {X 0,Y 502.837,Z 139.473,A -85,B 0,C 180,E1 -5698.371,E2 -5698.371} C_VEL
LIN {X 0,Y 502.793,Z 139.479,A -85,B 0,C 180,E1 -5701.498,E2 -5701.498} C_VEL
LIN {X 0,Y 502.803,Z 139.476,A -85,B 0,C 180,E1 -5704.444,E2 -5704.444} C_VEL
LIN {X 0,Y 502.776,Z 139.482,A -85,B 0,C 180,E1 -5707.177,E2 -5707.177} C_VEL
LIN {X 0,Y 502.782,Z 139.469,A -85,B 0,C 180,E1 -5710.014,E2 -5710.014} C_VEL
LIN {X 0,Y 502.796,Z 139.476,A -85,B 0,C 180,E1 -5712.198,E2 -5712.198} C_VEL
LIN {X 0,Y 502.794,Z 139.482,A -85,B 0,C 180,E1 -5715.467,E2 -5715.467} C_VEL
LIN {X 0,Y 502.819,Z 139.477,A -85,B 0,C 180,E1 -5719.003,E2 -5719.003} C_VEL
LIN {X 0,Y 502.789,Z 139.475,A -85,B 0,C 180,E1 -5722.046,E2 -5722.046} C_VEL
LIN {X 0,Y 502.801,Z 139.478,A -85,B 0,C 180,E1 -5725.034,E2 -5725.034} C_VEL
LIN {X 0,Y 502.779,Z 139.478,A -85,B 0,C 180,E1 -5727.915,E2 -5727.915} C_VEL
LIN {X 0,Y 502.83,Z 139.468,A -85,B 0,C 180,E1 -5730.712,E2 -5730.712} C_VEL
LIN {X 0,Y 502.852,Z 139.47,A -85,B 0,C 180,E1 -5733.438,E2 -5733.438} C_VEL
LIN {X 0,Y 502.781,Z 139.473,A -85,B 0,C 180,E1 -5736.086,E2 -5736.086} C_VEL
LIN {X 0,Y 502.774,Z 139.483,A -85,B 0,C 180,E1 -5738.688,E2 -5738.688} C_VEL
LIN {X 0,Y 502.82,Z 139.473,A -85,B 0,C 180,E1 -5741.248,E2 -5741.248} C_VEL
LIN {X 0,Y 502.814,Z 139.473,A -85,B 0,C 180,E1 -5743.767,E2 -5743.767} C_VEL
LIN {X 0,Y 502.825,Z 139.469,A -85,B 0,C 180,E1 -5746.254,E2 -5746.254} C_VEL
LIN {X 0,Y 502.871,Z 139.468,A -85,B 0,C 180,E1 -5748.717,E2 -5748.717} C_VEL
LIN {X 0,Y 502.891,Z 139.462,A -85,B 0,C 180,E1 -5751.966,E2 -5751.966} C_VEL
LIN {X 0,Y 502.929,Z 139.454,A -85,B 0,C 180,E1 -5754.386,E2 -5754.386} C_VEL
LIN {X 0,Y 503.014,Z 139.448,A -85,B 0,C 180,E1 -5757.598,E2 -5757.598} C_VEL
LIN {X 0,Y 503.014,Z 139.442,A -85,B 0,C 180,E1 -5760,E2 -5760} C_VEL
LIN {X 0,Y 503.014,Z 139.45,A -85,B 0,C 180,E1 -5762.402,E2 -5762.402} C_VEL
LIN {X 0,Y 502.929,Z 139.454,A -85,B 0,C 180,E1 -5765.614,E2 -5765.614} C_VEL
LIN {X 0,Y 502.891,Z 139.459,A -85,B 0,C 180,E1 -5768.033,E2 -5768.033} C_VEL
LIN {X 0,Y 502.87,Z 139.463,A -85,B 0,C 180,E1 -5771.283,E2 -5771.283} C_VEL
LIN {X 0,Y 502.841,Z 139.472,A -85,B 0,C 180,E1 -5774.571,E2 -5774.571} C_VEL
LIN {X 0,Y 502.851,Z 139.467,A -85,B 0,C 180,E1 -5777.907,E2 -5777.907} C_VEL
LIN {X 0,Y 502.82,Z 139.477,A -85,B 0,C 180,E1 -5780.537,E2 -5780.537} C_VEL
LIN {X 0,Y 502.795,Z 139.473,A -85,B 0,C 180,E1 -5783.04,E2 -5783.04} C_VEL
LIN {X 0,Y 502.83,Z 139.468,A -85,B 0,C 180,E1 -5785.676,E2 -5785.676} C_VEL
LIN {X 0,Y 502.83,Z 139.474,A -85,B 0,C 180,E1 -5788.373,E2 -5788.373} C_VEL
LIN {X 0,Y 502.786,Z 139.477,A -85,B 0,C 180,E1 -5791.5,E2 -5791.5} C_VEL
LIN {X 0,Y 502.797,Z 139.478,A -85,B 0,C 180,E1 -5794.445,E2 -5794.445} C_VEL
LIN {X 0,Y 502.772,Z 139.478,A -85,B 0,C 180,E1 -5797.179,E2 -5797.179} C_VEL
LIN {X 0,Y 502.779,Z 139.467,A -85,B 0,C 180,E1 -5800.016,E2 -5800.016} C_VEL
LIN {X 0,Y 502.794,Z 139.475,A -85,B 0,C 180,E1 -5802.2,E2 -5802.2} C_VEL
LIN {X 0,Y 502.793,Z 139.478,A -85,B 0,C 180,E1 -5805.469,E2 -5805.469} C_VEL
LIN {X 0,Y 502.828,Z 139.478,A -85,B 0,C 180,E1 -5807.866,E2 -5807.866} C_VEL
LIN {X 0,Y 502.803,Z 139.474,A -85,B 0,C 180,E1 -5811.026,E2 -5811.026} C_VEL
LIN {X 0,Y 502.778,Z 139.48,A -85,B 0,C 180,E1 -5814.169,E2 -5814.169} C_VEL
LIN {X 0,Y 502.827,Z 139.472,A -85,B 0,C 180,E1 -5816.994,E2 -5816.994} C_VEL
LIN {X 0,Y 502.822,Z 139.602,A -85,B 0,C 180,E1 -5817.94,E2 -5817.94} C_VEL
LIN {X 0,Y 508.869,Z 159.671,A -85,B 0,C 180,E1 -5820.312,E2 -5820.312} C_VEL
LIN {X 0,Y 509.089,Z 161.813,A -85,B 0,C 180,E1 -5820.536,E2 -5820.536} C_VEL
LIN {X 0,Y 507.619,Z 194.115,A -85,B 0,C 180,E1 -5823.593,E2 -5823.593} C_VEL
LIN {X 0,Y 506.229,Z 229.165,A -85,B 0,C 180,E1 -5826.831,E2 -5826.831} C_VEL
LIN {X 0,Y 505.849,Z 241.109,A -85,B 0,C 180,E1 -5827.902,E2 -5827.902} C_VEL
LIN {X 0,Y 507.823,Z 256.742,A -85,B 0,C 180,E1 -5828.223,E2 -5828.223} C_VEL
LIN {X 0,Y 506.655,Z 407.797,A -85,B 0,C 180,E1 -5830.424,E2 -5830.424} C_VEL
LIN {X 0,Y 506.265,Z 423.877,A -85,B 0,C 180,E1 -5830.829,E2 -5830.829} C_VEL
LIN {X 0,Y 505.824,Z 438.544,A -85,B 0,C 180,E1 -5831.365,E2 -5831.365} C_VEL
LIN {X 0,Y 505.266,Z 453.283,A -85,B 0,C 180,E1 -5832.078,E2 -5832.078} C_VEL
LIN {X 0,Y 504.762,Z 466.698,A -85,B 0,C 180,E1 -5832.896,E2 -5832.896} C_VEL
LIN {X 0,Y 504.206,Z 480.165,A -85,B 0,C 180,E1 -5833.903,E2 -5833.903} C_VEL
LIN {X 0,Y 503.658,Z 492.724,A -85,B 0,C 180,E1 -5835.041,E2 -5835.041} C_VEL
LIN {X 0,Y 503.209,Z 504.023,A -85,B 0,C 180,E1 -5836.266,E2 -5836.266} C_VEL
LIN {X 0,Y 502.928,Z 513.739,A -85,B 0,C 180,E1 -5837.492,E2 -5837.492} C_VEL
LIN {X 0,Y 502.671,Z 523.25,A -85,B 0,C 180,E1 -5838.917,E2 -5838.917} C_VEL
LIN {X 0,Y 502.418,Z 531.128,A -85,B 0,C 180,E1 -5840.338,E2 -5840.338} C_VEL
LIN {X 0,Y 502.327,Z 538.486,A -85,B 0,C 180,E1 -5841.959,E2 -5841.959} C_VEL
LIN {X 0,Y 502.3,Z 544.268,A -85,B 0,C 180,E1 -5843.574,E2 -5843.574} C_VEL
LIN {X 0,Y 502.248,Z 548.626,A -85,B 0,C 180,E1 -5845.185,E2 -5845.185} C_VEL
LIN {X 0,Y 502.243,Z 551.676,A -85,B 0,C 180,E1 -5846.792,E2 -5846.792} C_VEL
LIN {X 0,Y 502.167,Z 553.471,A -85,B 0,C 180,E1 -5848.397,E2 -5848.397} C_VEL
LIN {X 0,Y 502.213,Z 554.066,A -85,B 0,C 180,E1 -5850.001,E2 -5850.001} C_VEL
LIN {X 0,Y 502.176,Z 553.394,A -85,B 0,C 180,E1 -5851.605,E2 -5851.605} C_VEL
LIN {X 0,Y 502.257,Z 551.524,A -85,B 0,C 180,E1 -5853.21,E2 -5853.21} C_VEL
LIN {X 0,Y 502.27,Z 548.397,A -85,B 0,C 180,E1 -5854.817,E2 -5854.817} C_VEL
LIN {X 0,Y 502.302,Z 543.945,A -85,B 0,C 180,E1 -5856.428,E2 -5856.428} C_VEL
LIN {X 0,Y 502.387,Z 538.053,A -85,B 0,C 180,E1 -5858.043,E2 -5858.043} C_VEL
LIN {X 0,Y 502.51,Z 529.635,A -85,B 0,C 180,E1 -5859.866,E2 -5859.866} C_VEL
LIN {X 0,Y 502.713,Z 521.637,A -85,B 0,C 180,E1 -5861.288,E2 -5861.288} C_VEL
LIN {X 0,Y 502.935,Z 512.017,A -85,B 0,C 180,E1 -5862.715,E2 -5862.715} C_VEL
LIN {X 0,Y 503.292,Z 502.22,A -85,B 0,C 180,E1 -5863.939,E2 -5863.939} C_VEL
LIN {X 0,Y 503.757,Z 490.572,A -85,B 0,C 180,E1 -5865.165,E2 -5865.165} C_VEL
LIN {X 0,Y 504.271,Z 477.737,A -85,B 0,C 180,E1 -5866.29,E2 -5866.29} C_VEL
LIN {X 0,Y 504.795,Z 465.087,A -85,B 0,C 180,E1 -5867.21,E2 -5867.21} C_VEL
LIN {X 0,Y 505.354,Z 451.322,A -85,B 0,C 180,E1 -5868.026,E2 -5868.026} C_VEL
LIN {X 0,Y 505.904,Z 436.881,A -85,B 0,C 180,E1 -5868.701,E2 -5868.701} C_VEL
LIN {X 0,Y 506.342,Z 421.489,A -85,B 0,C 180,E1 -5869.24,E2 -5869.24} C_VEL
LIN {X 0,Y 506.67,Z 407.68,A -85,B 0,C 180,E1 -5869.578,E2 -5869.578} C_VEL
LIN {X 0,Y 507.776,Z 264.894,A -85,B 0,C 180,E1 -5871.658,E2 -5871.658} C_VEL
LIN {X 0,Y 507.645,Z 255.169,A -85,B 0,C 180,E1 -5871.808,E2 -5871.808} C_VEL
LIN {X 0,Y 505.683,Z 239.053,A -85,B 0,C 180,E1 -5872.148,E2 -5872.148} C_VEL
LIN {X 0,Y 506.806,Z 207.976,A -85,B 0,C 180,E1 -5875.022,E2 -5875.022} C_VEL
LIN {X 0,Y 508.273,Z 178.215,A -85,B 0,C 180,E1 -5877.89,E2 -5877.89} C_VEL
LIN {X 0,Y 509.306,Z 161.058,A -85,B 0,C 180,E1 -5879.617,E2 -5879.617} C_VEL
LIN {X 0,Y 506.676,Z 151.244,A -85,B 0,C 180,E1 -5880.879,E2 -5880.879} C_VEL
LIN {X 0,Y 502.844,Z 139.478,A -85,B 0,C 180,E1 -5882.583,E2 -5882.583} C_VEL
LIN {X 0,Y 502.773,Z 139.486,A -85,B 0,C 180,E1 -5885.831,E2 -5885.831} C_VEL
LIN {X 0,Y 502.794,Z 139.481,A -85,B 0,C 180,E1 -5888.978,E2 -5888.978} C_VEL
LIN {X 0,Y 502.747,Z 139.486,A -85,B 0,C 180,E1 -5892.192,E2 -5892.192} C_VEL
LIN {X 0,Y 502.78,Z 139.484,A -85,B 0,C 180,E1 -5895.472,E2 -5895.472} C_VEL
LIN {X 0,Y 502.751,Z 139.487,A -85,B 0,C 180,E1 -5898.927,E2 -5898.927} C_VEL
LIN {X 0,Y 502.756,Z 139.484,A -85,B 0,C 180,E1 -5902.043,E2 -5902.043} C_VEL
LIN {X 0,Y 502.785,Z 139.484,A -85,B 0,C 180,E1 -5905.033,E2 -5905.033} C_VEL
LIN {X 0,Y 502.761,Z 139.485,A -85,B 0,C 180,E1 -5907.914,E2 -5907.914} C_VEL
LIN {X 0,Y 502.794,Z 139.484,A -85,B 0,C 180,E1 -5910.71,E2 -5910.71} C_VEL
LIN {X 0,Y 502.801,Z 139.609,A -85,B 0,C 180,E1 -5912.926,E2 -5912.926} C_VEL
LIN {X 0,Y 505.467,Z 149.408,A -85,B 0,C 180,E1 -5914.967,E2 -5914.967} C_VEL
LIN {X 0,Y 506.975,Z 156.967,A -85,B 0,C 180,E1 -5916.444,E2 -5916.444} C_VEL
LIN {X 0,Y 506.112,Z 173.459,A -85,B 0,C 180,E1 -5919.262,E2 -5919.262} C_VEL
LIN {X 0,Y 505.223,Z 192.208,A -85,B 0,C 180,E1 -5922.389,E2 -5922.389} C_VEL
LIN {X 0,Y 504.944,Z 200.636,A -85,B 0,C 180,E1 -5923.742,E2 -5923.742} C_VEL
LIN {X 0,Y 506.813,Z 209.456,A -85,B 0,C 180,E1 -5924.002,E2 -5924.002} C_VEL
LIN {X 0,Y 505.288,Z 304.204,A -85,B 0,C 180,E1 -5925.707,E2 -5925.707} C_VEL
LIN {X 0,Y 505.183,Z 317.927,A -85,B 0,C 180,E1 -5926.012,E2 -5926.012} C_VEL
LIN {X 0,Y 504.991,Z 331.007,A -85,B 0,C 180,E1 -5926.469,E2 -5926.469} C_VEL
LIN {X 0,Y 504.788,Z 343.24,A -85,B 0,C 180,E1 -5927.058,E2 -5927.058} C_VEL
LIN {X 0,Y 504.444,Z 354.952,A -85,B 0,C 180,E1 -5927.79,E2 -5927.79} C_VEL
LIN {X 0,Y 504.158,Z 365.738,A -85,B 0,C 180,E1 -5928.644,E2 -5928.644} C_VEL
LIN {X 0,Y 503.885,Z 375.087,A -85,B 0,C 180,E1 -5929.553,E2 -5929.553} C_VEL
LIN {X 0,Y 503.644,Z 383.626,A -85,B 0,C 180,E1 -5930.563,E2 -5930.563} C_VEL
LIN {X 0,Y 503.279,Z 391.922,A -85,B 0,C 180,E1 -5931.771,E2 -5931.771} C_VEL
LIN {X 0,Y 503.042,Z 398.95,A -85,B 0,C 180,E1 -5933.057,E2 -5933.057} C_VEL
LIN {X 0,Y 502.863,Z 404.636,A -85,B 0,C 180,E1 -5934.386,E2 -5934.386} C_VEL
LIN {X 0,Y 502.728,Z 408.555,A -85,B 0,C 180,E1 -5935.59,E2 -5935.59} C_VEL
LIN {X 0,Y 502.607,Z 411.422,A -85,B 0,C 180,E1 -5936.794,E2 -5936.794} C_VEL
LIN {X 0,Y 502.589,Z 412.794,A -85,B 0,C 180,E1 -5937.596,E2 -5937.596} C_VEL
LIN {X 0,Y 502.616,Z 413.725,A -85,B 0,C 180,E1 -5938.398,E2 -5938.398} C_VEL
LIN {X 0,Y 502.538,Z 414.449,A -85,B 0,C 180,E1 -5940,E2 -5940} C_VEL
LIN {X 0,Y 502.552,Z 414.196,A -85,B 0,C 180,E1 -5940.801,E2 -5940.801} C_VEL
LIN {X 0,Y 502.487,Z 413.539,A -85,B 0,C 180,E1 -5941.603,E2 -5941.603} C_VEL
LIN {X 0,Y 502.58,Z 412.476,A -85,B 0,C 180,E1 -5942.404,E2 -5942.404} C_VEL
LIN {X 0,Y 502.529,Z 411.04,A -85,B 0,C 180,E1 -5943.207,E2 -5943.207} C_VEL
LIN {X 0,Y 502.681,Z 408.012,A -85,B 0,C 180,E1 -5944.41,E2 -5944.41} C_VEL
LIN {X 0,Y 502.669,Z 403.98,A -85,B 0,C 180,E1 -5945.617,E2 -5945.617} C_VEL
LIN {X 0,Y 502.911,Z 398.695,A -85,B 0,C 180,E1 -5946.84,E2 -5946.84} C_VEL
LIN {X 0,Y 503.077,Z 392.254,A -85,B 0,C 180,E1 -5948.031,E2 -5948.031} C_VEL
LIN {X 0,Y 503.304,Z 384.116,A -85,B 0,C 180,E1 -5949.241,E2 -5949.241} C_VEL
LIN {X 0,Y 503.559,Z 375.824,A -85,B 0,C 180,E1 -5950.25,E2 -5950.25} C_VEL
LIN {X 0,Y 503.836,Z 365.715,A -85,B 0,C 180,E1 -5951.262,E2 -5951.262} C_VEL
LIN {X 0,Y 504.218,Z 354.043,A -85,B 0,C 180,E1 -5952.188,E2 -5952.188} C_VEL
LIN {X 0,Y 504.483,Z 341.379,A -85,B 0,C 180,E1 -5952.982,E2 -5952.982} C_VEL
LIN {X 0,Y 504.676,Z 328.34,A -85,B 0,C 180,E1 -5953.592,E2 -5953.592} C_VEL
LIN {X 0,Y 504.923,Z 314.54,A -85,B 0,C 180,E1 -5954.047,E2 -5954.047} C_VEL
LIN {X 0,Y 505.072,Z 300.587,A -85,B 0,C 180,E1 -5954.325,E2 -5954.325} C_VEL
LIN {X 0,Y 505.803,Z 207.243,A -85,B 0,C 180,E1 -5955.8,E2 -5955.8} C_VEL
LIN {X 0,Y 503.914,Z 197.511,A -85,B 0,C 180,E1 -5956.038,E2 -5956.038} C_VEL
LIN {X 0,Y 504.522,Z 176.894,A -85,B 0,C 180,E1 -5959.32,E2 -5959.32} C_VEL
LIN {X 0,Y 505.139,Z 158.497,A -85,B 0,C 180,E1 -5962.28,E2 -5962.28} C_VEL
LIN {X 0,Y 505.294,Z 150.953,A -85,B 0,C 180,E1 -5963.511,E2 -5963.511} C_VEL
LIN {X 0,Y 502.833,Z 139.479,A -85,B 0,C 180,E1 -5965.565,E2 -5965.565} C_VEL
LIN {X 0,Y 502.8,Z 139.478,A -85,B 0,C 180,E1 -5968.375,E2 -5968.375} C_VEL
LIN {X 0,Y 502.799,Z 139.481,A -85,B 0,C 180,E1 -5971.143,E2 -5971.143} C_VEL
LIN {X 0,Y 502.808,Z 139.476,A -85,B 0,C 180,E1 -5973.994,E2 -5973.994} C_VEL
LIN {X 0,Y 502.769,Z 139.486,A -85,B 0,C 180,E1 -5977.175,E2 -5977.175} C_VEL
LIN {X 0,Y 502.792,Z 139.479,A -85,B 0,C 180,E1 -5979.145,E2 -5979.145} C_VEL
LIN {X 0,Y 502.112,Z 139.559,A -85,B 0,C 180,E1 -5979.813,E2 -5979.813} C_VEL
LIN {X 0,Y 499.265,Z 139.916,A -85,B 0,C 180,E1 -5980.9,E2 -5980.9} C_VEL
LIN {X 0,Y 496.861,Z 140.217,A -85,B 0,C 180,E1 -5981.775,E2 -5981.775} C_VEL
LIN {X 0,Y 495.819,Z 140.346,A -85,B 0,C 180,E1 -5982.45,E2 -5982.45} C_VEL
LIN {X 0,Y 495.728,Z 140.359,A -85,B 0,C 180,E1 -5982.679,E2 -5982.679} C_VEL
LIN {X 0,Y 495.733,Z 140.356,A -85,B 0,C 180,E1 -5985.998,E2 -5985.998} C_VEL
LIN {X 0,Y 495.77,Z 140.353,A -85,B 0,C 180,E1 -5989.3,E2 -5989.3} C_VEL
LIN {X 0,Y 495.733,Z 140.36,A -85,B 0,C 180,E1 -5992.438,E2 -5992.438} C_VEL
LIN {X 0,Y 495.775,Z 140.354,A -85,B 0,C 180,E1 -5995.456,E2 -5995.456} C_VEL
LIN {X 0,Y 495.759,Z 140.358,A -85,B 0,C 180,E1 -5998.363,E2 -5998.363} C_VEL
LIN {X 0,Y 495.79,Z 140.352,A -85,B 0,C 180,E1 -6001.507,E2 -6001.507} C_VEL
LIN {X 0,Y 495.82,Z 140.386,A -85,B 0,C 180,E1 -6004.159,E2 -6004.159} C_VEL
LIN {X 0,Y 498.777,Z 153.811,A -85,B 0,C 180,E1 -6006.331,E2 -6006.331} C_VEL
LIN {X 0,Y 498.928,Z 160.988,A -85,B 0,C 180,E1 -6007.323,E2 -6007.323} C_VEL
LIN {X 0,Y 502.351,Z 176.204,A -85,B 0,C 180,E1 -6007.734,E2 -6007.734} C_VEL
LIN {X 0,Y 500.966,Z 327.406,A -85,B 0,C 180,E1 -6009.984,E2 -6009.984} C_VEL
LIN {X 0,Y 500.755,Z 342.444,A -85,B 0,C 180,E1 -6010.368,E2 -6010.368} C_VEL
LIN {X 0,Y 500.347,Z 356.669,A -85,B 0,C 180,E1 -6010.885,E2 -6010.885} C_VEL
LIN {X 0,Y 499.926,Z 370.678,A -85,B 0,C 180,E1 -6011.559,E2 -6011.559} C_VEL
LIN {X 0,Y 499.308,Z 384.303,A -85,B 0,C 180,E1 -6012.384,E2 -6012.384} C_VEL
LIN {X 0,Y 498.662,Z 397.039,A -85,B 0,C 180,E1 -6013.333,E2 -6013.333} C_VEL
LIN {X 0,Y 498.122,Z 407.387,A -85,B 0,C 180,E1 -6014.248,E2 -6014.248} C_VEL
LIN {X 0,Y 497.496,Z 419.048,A -85,B 0,C 180,E1 -6015.477,E2 -6015.477} C_VEL
LIN {X 0,Y 496.932,Z 428.899,A -85,B 0,C 180,E1 -6016.713,E2 -6016.713} C_VEL
LIN {X 0,Y 496.416,Z 438.523,A -85,B 0,C 180,E1 -6018.155,E2 -6018.155} C_VEL
LIN {X 0,Y 496.009,Z 446.48,A -85,B 0,C 180,E1 -6019.591,E2 -6019.591} C_VEL
LIN {X 0,Y 495.733,Z 453.068,A -85,B 0,C 180,E1 -6021.027,E2 -6021.027} C_VEL
LIN {X 0,Y 495.464,Z 459.165,A -85,B 0,C 180,E1 -6022.665,E2 -6022.665} C_VEL
LIN {X 0,Y 495.261,Z 463.881,A -85,B 0,C 180,E1 -6024.298,E2 -6024.298} C_VEL
LIN {X 0,Y 495.237,Z 467.332,A -85,B 0,C 180,E1 -6025.93,E2 -6025.93} C_VEL
LIN {X 0,Y 495.074,Z 469.623,A -85,B 0,C 180,E1 -6027.558,E2 -6027.558} C_VEL
LIN {X 0,Y 494.989,Z 470.79,A -85,B 0,C 180,E1 -6029.185,E2 -6029.185} C_VEL
LIN {X 0,Y 494.989,Z 470.807,A -85,B 0,C 180,E1 -6030.812,E2 -6030.812} C_VEL
LIN {X 0,Y 495.073,Z 469.706,A -85,B 0,C 180,E1 -6032.44,E2 -6032.44} C_VEL
LIN {X 0,Y 495.224,Z 467.487,A -85,B 0,C 180,E1 -6034.068,E2 -6034.068} C_VEL
LIN {X 0,Y 495.253,Z 464.115,A -85,B 0,C 180,E1 -6035.7,E2 -6035.7} C_VEL
LIN {X 0,Y 495.457,Z 459.477,A -85,B 0,C 180,E1 -6037.334,E2 -6037.334} C_VEL
LIN {X 0,Y 495.728,Z 453.455,A -85,B 0,C 180,E1 -6038.971,E2 -6038.971} C_VEL
LIN {X 0,Y 496.023,Z 445.88,A -85,B 0,C 180,E1 -6040.613,E2 -6040.613} C_VEL
LIN {X 0,Y 496.453,Z 437.81,A -85,B 0,C 180,E1 -6042.048,E2 -6042.048} C_VEL
LIN {X 0,Y 496.983,Z 428.026,A -85,B 0,C 180,E1 -6043.492,E2 -6043.492} C_VEL
LIN {X 0,Y 497.533,Z 418.045,A -85,B 0,C 180,E1 -6044.729,E2 -6044.729} C_VEL
LIN {X 0,Y 498.184,Z 406.262,A -85,B 0,C 180,E1 -6045.949,E2 -6045.949} C_VEL
LIN {X 0,Y 498.886,Z 392.869,A -85,B 0,C 180,E1 -6047.09,E2 -6047.09} C_VEL
LIN {X 0,Y 499.562,Z 379.337,A -85,B 0,C 180,E1 -6048.028,E2 -6048.028} C_VEL
LIN {X 0,Y 500.043,Z 365.46,A -85,B 0,C 180,E1 -6048.806,E2 -6048.806} C_VEL
LIN {X 0,Y 500.515,Z 351.182,A -85,B 0,C 180,E1 -6049.426,E2 -6049.426} C_VEL
LIN {X 0,Y 500.836,Z 336.251,A -85,B 0,C 180,E1 -6049.903,E2 -6049.903} C_VEL
LIN {X 0,Y 501.081,Z 321.806,A -85,B 0,C 180,E1 -6050.209,E2 -6050.209} C_VEL
LIN {X 0,Y 502.388,Z 175.668,A -85,B 0,C 180,E1 -6052.364,E2 -6052.364} C_VEL
LIN {X 0,Y 498.936,Z 160.991,A -85,B 0,C 180,E1 -6052.772,E2 -6052.772} C_VEL
LIN {X 0,Y 498.762,Z 153.38,A -85,B 0,C 180,E1 -6053.823,E2 -6053.823} C_VEL
LIN {X 0,Y 495.812,Z 140.354,A -85,B 0,C 180,E1 -6055.952,E2 -6055.952} C_VEL
LIN {X 0,Y 495.768,Z 140.354,A -85,B 0,C 180,E1 -6058.814,E2 -6058.814} C_VEL
LIN {X 0,Y 495.755,Z 140.353,A -85,B 0,C 180,E1 -6061.725,E2 -6061.725} C_VEL
LIN {X 0,Y 495.773,Z 140.353,A -85,B 0,C 180,E1 -6064.694,E2 -6064.694} C_VEL
LIN {X 0,Y 495.727,Z 140.363,A -85,B 0,C 180,E1 -6067.56,E2 -6067.56} C_VEL
LIN {X 0,Y 495.761,Z 140.343,A -85,B 0,C 180,E1 -6070.699,E2 -6070.699} C_VEL
LIN {X 0,Y 495.728,Z 140.357,A -85,B 0,C 180,E1 -6073.694,E2 -6073.694} C_VEL
LIN {X 0,Y 495.721,Z 140.357,A -85,B 0,C 180,E1 -6076.304,E2 -6076.304} C_VEL
LIN {X 0,Y 495.773,Z 140.358,A -85,B 0,C 180,E1 -6079.301,E2 -6079.301} C_VEL
LIN {X 0,Y 495.756,Z 140.355,A -85,B 0,C 180,E1 -6081.409,E2 -6081.409} C_VEL
LIN {X 0,Y 495.749,Z 140.353,A -85,B 0,C 180,E1 -6084.462,E2 -6084.462} C_VEL
LIN {X 0,Y 495.76,Z 140.357,A -85,B 0,C 180,E1 -6087.405,E2 -6087.405} C_VEL
LIN {X 0,Y 495.772,Z 140.344,A -85,B 0,C 180,E1 -6090.254,E2 -6090.254} C_VEL
LIN {X 0,Y 495.813,Z 140.349,A -85,B 0,C 180,E1 -6093.25,E2 -6093.25} C_VEL
LIN {X 0,Y 495.742,Z 140.351,A -85,B 0,C 180,E1 -6095.724,E2 -6095.724} C_VEL
LIN {X 0,Y 495.737,Z 140.356,A -85,B 0,C 180,E1 -6098.371,E2 -6098.371} C_VEL
LIN {X 0,Y 495.775,Z 140.349,A -85,B 0,C 180,E1 -6100.971,E2 -6100.971} C_VEL
LIN {X 0,Y 495.771,Z 140.352,A -85,B 0,C 180,E1 -6103.53,E2 -6103.53} C_VEL
LIN {X 0,Y 495.786,Z 140.345,A -85,B 0,C 180,E1 -6106.055,E2 -6106.055} C_VEL
LIN {X 0,Y 495.844,Z 140.34,A -85,B 0,C 180,E1 -6108.555,E2 -6108.555} C_VEL
LIN {X 0,Y 495.862,Z 140.337,A -85,B 0,C 180,E1 -6111.852,E2 -6111.852} C_VEL
LIN {X 0,Y 495.886,Z 140.33,A -85,B 0,C 180,E1 -6114.306,E2 -6114.306} C_VEL
LIN {X 0,Y 495.983,Z 140.324,A -85,B 0,C 180,E1 -6117.564,E2 -6117.564} C_VEL
LIN {X 0,Y 495.986,Z 140.317,A -85,B 0,C 180,E1 -6120,E2 -6120} C_VEL
LIN {X 0,Y 495.983,Z 140.326,A -85,B 0,C 180,E1 -6122.436,E2 -6122.436} C_VEL
LIN {X 0,Y 495.886,Z 140.331,A -85,B 0,C 180,E1 -6125.693,E2 -6125.693} C_VEL
LIN {X 0,Y 495.863,Z 140.335,A -85,B 0,C 180,E1 -6128.148,E2 -6128.148} C_VEL
LIN {X 0,Y 495.844,Z 140.337,A -85,B 0,C 180,E1 -6131.445,E2 -6131.445} C_VEL
LIN {X 0,Y 495.783,Z 140.351,A -85,B 0,C 180,E1 -6134.783,E2 -6134.783} C_VEL
LIN {X 0,Y 495.777,Z 140.346,A -85,B 0,C 180,E1 -6137.319,E2 -6137.319} C_VEL
LIN {X 0,Y 495.767,Z 140.346,A -85,B 0,C 180,E1 -6139.89,E2 -6139.89} C_VEL
LIN {X 0,Y 495.754,Z 140.352,A -85,B 0,C 180,E1 -6142.863,E2 -6142.863} C_VEL
LIN {X 0,Y 495.781,Z 140.35,A -85,B 0,C 180,E1 -6146.068,E2 -6146.068} C_VEL
LIN {X 0,Y 495.761,Z 140.349,A -85,B 0,C 180,E1 -6148.815,E2 -6148.815} C_VEL
LIN {X 0,Y 495.748,Z 140.355,A -85,B 0,C 180,E1 -6151.727,E2 -6151.727} C_VEL
LIN {X 0,Y 495.767,Z 140.352,A -85,B 0,C 180,E1 -6154.696,E2 -6154.696} C_VEL
LIN {X 0,Y 495.722,Z 140.357,A -85,B 0,C 180,E1 -6157.562,E2 -6157.562} C_VEL
LIN {X 0,Y 495.758,Z 140.341,A -85,B 0,C 180,E1 -6160.701,E2 -6160.701} C_VEL
LIN {X 0,Y 495.726,Z 140.363,A -85,B 0,C 180,E1 -6164.002,E2 -6164.002} C_VEL
LIN {X 0,Y 495.755,Z 140.353,A -85,B 0,C 180,E1 -6167.122,E2 -6167.122} C_VEL
LIN {X 0,Y 495.776,Z 140.353,A -85,B 0,C 180,E1 -6170.366,E2 -6170.366} C_VEL
LIN {X 0,Y 495.727,Z 140.356,A -85,B 0,C 180,E1 -6173.458,E2 -6173.458} C_VEL
LIN {X 0,Y 495.754,Z 140.353,A -85,B 0,C 180,E1 -6176.437,E2 -6176.437} C_VEL
LIN {X 0,Y 495.776,Z 140.52,A -85,B 0,C 180,E1 -6177.59,E2 -6177.59} C_VEL
LIN {X 0,Y 501.961,Z 160.926,A -85,B 0,C 180,E1 -6180.047,E2 -6180.047} C_VEL
LIN {X 0,Y 502.454,Z 162.78,A -85,B 0,C 180,E1 -6180.26,E2 -6180.26} C_VEL
LIN {X 0,Y 500.921,Z 194.65,A -85,B 0,C 180,E1 -6183.324,E2 -6183.324} C_VEL
LIN {X 0,Y 499.397,Z 229.795,A -85,B 0,C 180,E1 -6186.624,E2 -6186.624} C_VEL
LIN {X 0,Y 499.076,Z 240.192,A -85,B 0,C 180,E1 -6187.579,E2 -6187.579} C_VEL
LIN {X 0,Y 501.201,Z 258.877,A -85,B 0,C 180,E1 -6187.959,E2 -6187.959} C_VEL
LIN {X 0,Y 499.965,Z 407.346,A -85,B 0,C 180,E1 -6190.151,E2 -6190.151} C_VEL
LIN {X 0,Y 499.55,Z 423.322,A -85,B 0,C 180,E1 -6190.559,E2 -6190.559} C_VEL
LIN {X 0,Y 499.056,Z 438.006,A -85,B 0,C 180,E1 -6191.102,E2 -6191.102} C_VEL
LIN {X 0,Y 498.436,Z 452.729,A -85,B 0,C 180,E1 -6191.824,E2 -6191.824} C_VEL
LIN {X 0,Y 497.883,Z 466.134,A -85,B 0,C 180,E1 -6192.652,E2 -6192.652} C_VEL
LIN {X 0,Y 497.306,Z 479.841,A -85,B 0,C 180,E1 -6193.695,E2 -6193.695} C_VEL
LIN {X 0,Y 496.689,Z 492.145,A -85,B 0,C 180,E1 -6194.826,E2 -6194.826} C_VEL
LIN {X 0,Y 496.21,Z 503.441,A -85,B 0,C 180,E1 -6196.069,E2 -6196.069} C_VEL
LIN {X 0,Y 495.824,Z 514.407,A -85,B 0,C 180,E1 -6197.518,E2 -6197.518} C_VEL
LIN {X 0,Y 495.564,Z 523.525,A -85,B 0,C 180,E1 -6198.963,E2 -6198.963} C_VEL
LIN {X 0,Y 495.306,Z 532.104,A -85,B 0,C 180,E1 -6200.61,E2 -6200.61} C_VEL
LIN {X 0,Y 495.244,Z 539.086,A -85,B 0,C 180,E1 -6202.253,E2 -6202.253} C_VEL
LIN {X 0,Y 495.26,Z 544.545,A -85,B 0,C 180,E1 -6203.892,E2 -6203.892} C_VEL
LIN {X 0,Y 495.212,Z 547.667,A -85,B 0,C 180,E1 -6205.116,E2 -6205.116} C_VEL
LIN {X 0,Y 495.195,Z 550.724,A -85,B 0,C 180,E1 -6206.747,E2 -6206.747} C_VEL
LIN {X 0,Y 495.128,Z 552.519,A -85,B 0,C 180,E1 -6208.374,E2 -6208.374} C_VEL
LIN {X 0,Y 495.194,Z 553.11,A -85,B 0,C 180,E1 -6210.001,E2 -6210.001} C_VEL
LIN {X 0,Y 495.139,Z 552.423,A -85,B 0,C 180,E1 -6211.628,E2 -6211.628} C_VEL
LIN {X 0,Y 495.213,Z 550.533,A -85,B 0,C 180,E1 -6213.255,E2 -6213.255} C_VEL
LIN {X 0,Y 495.239,Z 547.378,A -85,B 0,C 180,E1 -6214.885,E2 -6214.885} C_VEL
LIN {X 0,Y 495.253,Z 542.748,A -85,B 0,C 180,E1 -6216.611,E2 -6216.611} C_VEL
LIN {X 0,Y 495.296,Z 537.329,A -85,B 0,C 180,E1 -6218.158,E2 -6218.158} C_VEL
LIN {X 0,Y 495.38,Z 530.074,A -85,B 0,C 180,E1 -6219.803,E2 -6219.803} C_VEL
LIN {X 0,Y 495.62,Z 522.306,A -85,B 0,C 180,E1 -6221.244,E2 -6221.244} C_VEL
LIN {X 0,Y 495.872,Z 512.944,A -85,B 0,C 180,E1 -6222.691,E2 -6222.691} C_VEL
LIN {X 0,Y 496.247,Z 503.429,A -85,B 0,C 180,E1 -6223.932,E2 -6223.932} C_VEL
LIN {X 0,Y 496.702,Z 492.122,A -85,B 0,C 180,E1 -6225.176,E2 -6225.176} C_VEL
LIN {X 0,Y 497.269,Z 479.793,A -85,B 0,C 180,E1 -6226.31,E2 -6226.31} C_VEL
LIN {X 0,Y 497.874,Z 466.106,A -85,B 0,C 180,E1 -6227.35,E2 -6227.35} C_VEL
LIN {X 0,Y 498.463,Z 452.703,A -85,B 0,C 180,E1 -6228.178,E2 -6228.178} C_VEL
LIN {X 0,Y 499.08,Z 437.949,A -85,B 0,C 180,E1 -6228.899,E2 -6228.899} C_VEL
LIN {X 0,Y 499.594,Z 422.167,A -85,B 0,C 180,E1 -6229.475,E2 -6229.475} C_VEL
LIN {X 0,Y 499.982,Z 407.221,A -85,B 0,C 180,E1 -6229.85,E2 -6229.85} C_VEL
LIN {X 0,Y 501.233,Z 257.783,A -85,B 0,C 180,E1 -6232.056,E2 -6232.056} C_VEL
LIN {X 0,Y 498.879,Z 238.407,A -85,B 0,C 180,E1 -6232.466,E2 -6232.466} C_VEL
LIN {X 0,Y 500.118,Z 207.607,A -85,B 0,C 180,E1 -6235.38,E2 -6235.38} C_VEL
LIN {X 0,Y 501.788,Z 178.195,A -85,B 0,C 180,E1 -6238.287,E2 -6238.287} C_VEL
LIN {X 0,Y 502.816,Z 163.652,A -85,B 0,C 180,E1 -6239.782,E2 -6239.782} C_VEL
LIN {X 0,Y 500.734,Z 155.36,A -85,B 0,C 180,E1 -6240.868,E2 -6240.868} C_VEL
LIN {X 0,Y 496.44,Z 142.512,A -85,B 0,C 180,E1 -6242.783,E2 -6242.783} C_VEL
LIN {X 0,Y 495.786,Z 140.355,A -85,B 0,C 180,E1 -6243.134,E2 -6243.134} C_VEL
LIN {X 0,Y 495.714,Z 140.365,A -85,B 0,C 180,E1 -6246.088,E2 -6246.088} C_VEL
LIN {X 0,Y 495.759,Z 140.357,A -85,B 0,C 180,E1 -6248.768,E2 -6248.768} C_VEL
LIN {X 0,Y 495.725,Z 140.363,A -85,B 0,C 180,E1 -6251.785,E2 -6251.785} C_VEL
LIN {X 0,Y 495.734,Z 140.362,A -85,B 0,C 180,E1 -6255.142,E2 -6255.142} C_VEL
LIN {X 0,Y 495.703,Z 140.362,A -85,B 0,C 180,E1 -6258.213,E2 -6258.213} C_VEL
LIN {X 0,Y 495.715,Z 140.364,A -85,B 0,C 180,E1 -6261.405,E2 -6261.405} C_VEL
LIN {X 0,Y 495.73,Z 140.361,A -85,B 0,C 180,E1 -6264.461,E2 -6264.461} C_VEL
LIN {X 0,Y 495.743,Z 140.361,A -85,B 0,C 180,E1 -6267.404,E2 -6267.404} C_VEL
LIN {X 0,Y 495.742,Z 140.361,A -85,B 0,C 180,E1 -6270.252,E2 -6270.252} C_VEL
LIN {X 0,Y 495.755,Z 140.552,A -85,B 0,C 180,E1 -6272.394,E2 -6272.394} C_VEL
LIN {X 0,Y 498.458,Z 150.115,A -85,B 0,C 180,E1 -6274.472,E2 -6274.472} C_VEL
LIN {X 0,Y 500.346,Z 158.683,A -85,B 0,C 180,E1 -6276.208,E2 -6276.208} C_VEL
LIN {X 0,Y 499.533,Z 173.366,A -85,B 0,C 180,E1 -6278.76,E2 -6278.76} C_VEL
LIN {X 0,Y 498.541,Z 192.055,A -85,B 0,C 180,E1 -6281.933,E2 -6281.933} C_VEL
LIN {X 0,Y 498.204,Z 201.133,A -85,B 0,C 180,E1 -6283.424,E2 -6283.424} C_VEL
LIN {X 0,Y 500.229,Z 210.106,A -85,B 0,C 180,E1 -6283.708,E2 -6283.708} C_VEL
LIN {X 0,Y 498.545,Z 302.146,A -85,B 0,C 180,E1 -6285.431,E2 -6285.431} C_VEL
LIN {X 0,Y 498.416,Z 317.695,A -85,B 0,C 180,E1 -6285.766,E2 -6285.766} C_VEL
LIN {X 0,Y 498.193,Z 331.052,A -85,B 0,C 180,E1 -6286.228,E2 -6286.228} C_VEL
LIN {X 0,Y 497.981,Z 344.027,A -85,B 0,C 180,E1 -6286.857,E2 -6286.857} C_VEL
LIN {X 0,Y 497.644,Z 355.092,A -85,B 0,C 180,E1 -6287.55,E2 -6287.55} C_VEL
LIN {X 0,Y 497.325,Z 365.655,A -85,B 0,C 180,E1 -6288.383,E2 -6288.383} C_VEL
LIN {X 0,Y 496.985,Z 376.135,A -85,B 0,C 180,E1 -6289.407,E2 -6289.407} C_VEL
LIN {X 0,Y 496.717,Z 384.665,A -85,B 0,C 180,E1 -6290.43,E2 -6290.43} C_VEL
LIN {X 0,Y 496.331,Z 392.97,A -85,B 0,C 180,E1 -6291.655,E2 -6291.655} C_VEL
LIN {X 0,Y 496.09,Z 399.985,A -85,B 0,C 180,E1 -6292.958,E2 -6292.958} C_VEL
LIN {X 0,Y 495.88,Z 405.676,A -85,B 0,C 180,E1 -6294.306,E2 -6294.306} C_VEL
LIN {X 0,Y 495.724,Z 409.591,A -85,B 0,C 180,E1 -6295.528,E2 -6295.528} C_VEL
LIN {X 0,Y 495.62,Z 412.448,A -85,B 0,C 180,E1 -6296.748,E2 -6296.748} C_VEL
LIN {X 0,Y 495.575,Z 413.818,A -85,B 0,C 180,E1 -6297.562,E2 -6297.562} C_VEL
LIN {X 0,Y 495.605,Z 414.742,A -85,B 0,C 180,E1 -6298.375,E2 -6298.375} C_VEL
LIN {X 0,Y 495.52,Z 415.447,A -85,B 0,C 180,E1 -6300,E2 -6300} C_VEL
LIN {X 0,Y 495.534,Z 415.182,A -85,B 0,C 180,E1 -6300.813,E2 -6300.813} C_VEL
LIN {X 0,Y 495.465,Z 414.513,A -85,B 0,C 180,E1 -6301.626,E2 -6301.626} C_VEL
LIN {X 0,Y 495.563,Z 413.431,A -85,B 0,C 180,E1 -6302.439,E2 -6302.439} C_VEL
LIN {X 0,Y 495.501,Z 411.975,A -85,B 0,C 180,E1 -6303.252,E2 -6303.252} C_VEL
LIN {X 0,Y 495.664,Z 408.915,A -85,B 0,C 180,E1 -6304.473,E2 -6304.473} C_VEL
LIN {X 0,Y 495.669,Z 404.845,A -85,B 0,C 180,E1 -6305.696,E2 -6305.696} C_VEL
LIN {X 0,Y 495.921,Z 399.574,A -85,B 0,C 180,E1 -6306.925,E2 -6306.925} C_VEL
LIN {X 0,Y 496.109,Z 393.025,A -85,B 0,C 180,E1 -6308.144,E2 -6308.144} C_VEL
LIN {X 0,Y 496.355,Z 384.839,A -85,B 0,C 180,E1 -6309.371,E2 -6309.371} C_VEL
LIN {X 0,Y 496.625,Z 376.494,A -85,B 0,C 180,E1 -6310.395,E2 -6310.395} C_VEL
LIN {X 0,Y 496.919,Z 366.324,A -85,B 0,C 180,E1 -6311.42,E2 -6311.42} C_VEL
LIN {X 0,Y 497.314,Z 354.696,A -85,B 0,C 180,E1 -6312.352,E2 -6312.352} C_VEL
LIN {X 0,Y 497.575,Z 343.635,A -85,B 0,C 180,E1 -6313.061,E2 -6313.061} C_VEL
LIN {X 0,Y 497.826,Z 331.273,A -85,B 0,C 180,E1 -6313.678,E2 -6313.678} C_VEL
LIN {X 0,Y 497.978,Z 319.295,A -85,B 0,C 180,E1 -6314.116,E2 -6314.116} C_VEL
LIN {X 0,Y 498.159,Z 305.321,A -85,B 0,C 180,E1 -6314.45,E2 -6314.45} C_VEL
LIN {X 0,Y 499.022,Z 208.231,A -85,B 0,C 180,E1 -6316.022,E2 -6316.022} C_VEL
LIN {X 0,Y 497.023,Z 197.695,A -85,B 0,C 180,E1 -6316.295,E2 -6316.295} C_VEL
LIN {X 0,Y 497.663,Z 177.132,A -85,B 0,C 180,E1 -6319.597,E2 -6319.597} C_VEL
LIN {X 0,Y 498.279,Z 158.666,A -85,B 0,C 180,E1 -6322.603,E2 -6322.603} C_VEL
LIN {X 0,Y 498.445,Z 152.71,A -85,B 0,C 180,E1 -6323.58,E2 -6323.58} C_VEL
LIN {X 0,Y 495.813,Z 140.353,A -85,B 0,C 180,E1 -6325.813,E2 -6325.813} C_VEL
LIN {X 0,Y 495.748,Z 140.357,A -85,B 0,C 180,E1 -6328.816,E2 -6328.816} C_VEL
LIN {X 0,Y 495.759,Z 140.357,A -85,B 0,C 180,E1 -6331.725,E2 -6331.725} C_VEL
LIN {X 0,Y 495.772,Z 140.352,A -85,B 0,C 180,E1 -6334.693,E2 -6334.693} C_VEL
LIN {X 0,Y 495.726,Z 140.361,A -85,B 0,C 180,E1 -6337.562,E2 -6337.562} C_VEL
LIN {X 0,Y 495.76,Z 140.348,A -85,B 0,C 180,E1 -6340.046,E2 -6340.046} C_VEL
LIN {X 0,Y 495.728,Z 140.359,A -85,B 0,C 180,E1 -6342.679,E2 -6342.679} C_VEL
LIN {X 0,Y 495.047,Z 140.448,A -85,B 0,C 180,E1 -6343.358,E2 -6343.358} C_VEL
LIN {X 0,Y 492.198,Z 140.801,A -85,B 0,C 180,E1 -6344.46,E2 -6344.46} C_VEL
LIN {X 0,Y 489.799,Z 141.099,A -85,B 0,C 180,E1 -6345.348,E2 -6345.348} C_VEL
LIN {X 0,Y 488.772,Z 141.223,A -85,B 0,C 180,E1 -6346.033,E2 -6346.033} C_VEL
LIN {X 0,Y 488.689,Z 141.234,A -85,B 0,C 180,E1 -6346.266,E2 -6346.266} C_VEL
LIN {X 0,Y 488.712,Z 141.234,A -85,B 0,C 180,E1 -6348.584,E2 -6348.584} C_VEL
LIN {X 0,Y 488.705,Z 141.238,A -85,B 0,C 180,E1 -6350.947,E2 -6350.947} C_VEL
LIN {X 0,Y 488.682,Z 141.237,A -85,B 0,C 180,E1 -6353.867,E2 -6353.867} C_VEL
LIN {X 0,Y 488.74,Z 141.232,A -85,B 0,C 180,E1 -6356.876,E2 -6356.876} C_VEL
LIN {X 0,Y 488.727,Z 141.231,A -85,B 0,C 180,E1 -6359.78,E2 -6359.78} C_VEL
LIN {X 0,Y 488.796,Z 141.227,A -85,B 0,C 180,E1 -6363.056,E2 -6363.056} C_VEL
LIN {X 0,Y 488.773,Z 141.288,A -85,B 0,C 180,E1 -6363.873,E2 -6363.873} C_VEL
LIN {X 0,Y 491.913,Z 155.151,A -85,B 0,C 180,E1 -6366.117,E2 -6366.117} C_VEL
LIN {X 0,Y 492.197,Z 160.557,A -85,B 0,C 180,E1 -6366.879,E2 -6366.879} C_VEL
LIN {X 0,Y 492.179,Z 161.459,A -85,B 0,C 180,E1 -6366.994,E2 -6366.994} C_VEL
LIN {X 0,Y 495.793,Z 177.104,A -85,B 0,C 180,E1 -6367.429,E2 -6367.429} C_VEL
LIN {X 0,Y 494.352,Z 327.04,A -85,B 0,C 180,E1 -6369.687,E2 -6369.687} C_VEL
LIN {X 0,Y 494.101,Z 342.131,A -85,B 0,C 180,E1 -6370.066,E2 -6370.066} C_VEL
LIN {X 0,Y 493.717,Z 355.991,A -85,B 0,C 180,E1 -6370.564,E2 -6370.564} C_VEL
LIN {X 0,Y 493.271,Z 369.344,A -85,B 0,C 180,E1 -6371.194,E2 -6371.194} C_VEL
LIN {X 0,Y 492.631,Z 383.355,A -85,B 0,C 180,E1 -6372.03,E2 -6372.03} C_VEL
LIN {X 0,Y 491.982,Z 396.119,A -85,B 0,C 180,E1 -6372.971,E2 -6372.971} C_VEL
LIN {X 0,Y 491.311,Z 408.038,A -85,B 0,C 180,E1 -6374.031,E2 -6374.031} C_VEL
LIN {X 0,Y 490.63,Z 419.627,A -85,B 0,C 180,E1 -6375.269,E2 -6375.269} C_VEL
LIN {X 0,Y 490.055,Z 429.478,A -85,B 0,C 180,E1 -6376.523,E2 -6376.523} C_VEL
LIN {X 0,Y 489.48,Z 439.23,A -85,B 0,C 180,E1 -6378.005,E2 -6378.005} C_VEL
LIN {X 0,Y 488.979,Z 448.089,A -85,B 0,C 180,E1 -6379.649,E2 -6379.649} C_VEL
LIN {X 0,Y 488.64,Z 455.332,A -85,B 0,C 180,E1 -6381.313,E2 -6381.313} C_VEL
LIN {X 0,Y 488.424,Z 459.751,A -85,B 0,C 180,E1 -6382.558,E2 -6382.558} C_VEL
LIN {X 0,Y 488.21,Z 464.467,A -85,B 0,C 180,E1 -6384.216,E2 -6384.216} C_VEL
LIN {X 0,Y 488.174,Z 467.917,A -85,B 0,C 180,E1 -6385.871,E2 -6385.871} C_VEL
LIN {X 0,Y 488.013,Z 470.207,A -85,B 0,C 180,E1 -6387.523,E2 -6387.523} C_VEL
LIN {X 0,Y 487.914,Z 471.375,A -85,B 0,C 180,E1 -6389.174,E2 -6389.174} C_VEL
LIN {X 0,Y 487.914,Z 471.392,A -85,B 0,C 180,E1 -6390.824,E2 -6390.824} C_VEL
LIN {X 0,Y 488.013,Z 470.289,A -85,B 0,C 180,E1 -6392.475,E2 -6392.475} C_VEL
LIN {X 0,Y 488.162,Z 468.07,A -85,B 0,C 180,E1 -6394.127,E2 -6394.127} C_VEL
LIN {X 0,Y 488.201,Z 464.697,A -85,B 0,C 180,E1 -6395.782,E2 -6395.782} C_VEL
LIN {X 0,Y 488.414,Z 460.059,A -85,B 0,C 180,E1 -6397.44,E2 -6397.44} C_VEL
LIN {X 0,Y 488.708,Z 454.035,A -85,B 0,C 180,E1 -6399.101,E2 -6399.101} C_VEL
LIN {X 0,Y 489.059,Z 446.458,A -85,B 0,C 180,E1 -6400.766,E2 -6400.766} C_VEL
LIN {X 0,Y 489.513,Z 438.451,A -85,B 0,C 180,E1 -6402.211,E2 -6402.211} C_VEL
LIN {X 0,Y 490.084,Z 428.599,A -85,B 0,C 180,E1 -6403.686,E2 -6403.686} C_VEL
LIN {X 0,Y 490.69,Z 418.615,A -85,B 0,C 180,E1 -6404.939,E2 -6404.939} C_VEL
LIN {X 0,Y 491.377,Z 406.971,A -85,B 0,C 180,E1 -6406.163,E2 -6406.163} C_VEL
LIN {X 0,Y 492.05,Z 394.935,A -85,B 0,C 180,E1 -6407.217,E2 -6407.217} C_VEL
LIN {X 0,Y 492.74,Z 381.583,A -85,B 0,C 180,E1 -6408.179,E2 -6408.179} C_VEL
LIN {X 0,Y 493.317,Z 367.073,A -85,B 0,C 180,E1 -6409.018,E2 -6409.018} C_VEL
